LIN {X 0,Y 461.687,Z 311.629,A -85,B 0,C 180,E1 20728.292,E2 20728.292} C_VEL
LIN {X 0,Y 456.016,Z 403.282,A -85,B 0,C 180,E1 20726.276,E2 20726.276} C_VEL
LIN {X 0,Y 452.13,Z 492.328,A -85,B 0,C 180,E1 20724.472,E2 20724.472} C_VEL
LIN {X 0,Y 450.29,Z 542.964,A -85,B 0,C 180,E1 20723.46,E2 20723.46} C_VEL
LIN {X 0,Y 449.055,Z 565.43,A -85,B 0,C 180,E1 20722.774,E2 20722.774} C_VEL
LIN {X 0,Y 447.46,Z 585.999,A -85,B 0,C 180,E1 20721.912,E2 20721.912} C_VEL
LIN {X 0,Y 445.534,Z 606.342,A -85,B 0,C 180,E1 20720.838,E2 20720.838} C_VEL
LIN {X 0,Y 443.351,Z 625.885,A -85,B 0,C 180,E1 20719.568,E2 20719.568} C_VEL
LIN {X 0,Y 440.916,Z 645.179,A -85,B 0,C 180,E1 20718.033,E2 20718.033} C_VEL
LIN {X 0,Y 438.41,Z 662.746,A -85,B 0,C 180,E1 20716.361,E2 20716.361} C_VEL
LIN {X 0,Y 435.747,Z 680.551,A -85,B 0,C 180,E1 20714.35,E2 20714.35} C_VEL
LIN {X 0,Y 433.448,Z 695.322,A -85,B 0,C 180,E1 20712.389,E2 20712.389} C_VEL
LIN {X 0,Y 431.176,Z 709.526,A -85,B 0,C 180,E1 20710.152,E2 20710.152} C_VEL
LIN {X 0,Y 429.165,Z 722.41,A -85,B 0,C 180,E1 20707.768,E2 20707.768} C_VEL
LIN {X 0,Y 427.471,Z 733.989,A -85,B 0,C 180,E1 20705.236,E2 20705.236} C_VEL
LIN {X 0,Y 426.053,Z 744.612,A -85,B 0,C 180,E1 20702.423,E2 20702.423} C_VEL
LIN {X 0,Y 425.075,Z 753.264,A -85,B 0,C 180,E1 20699.598,E2 20699.598} C_VEL
LIN {X 0,Y 424.433,Z 760.513,A -85,B 0,C 180,E1 20696.626,E2 20696.626} C_VEL
LIN {X 0,Y 424.108,Z 766.032,A -85,B 0,C 180,E1 20693.64,E2 20693.64} C_VEL
LIN {X 0,Y 423.956,Z 769.849,A -85,B 0,C 180,E1 20690.637,E2 20690.637} C_VEL
LIN {X 0,Y 423.908,Z 772.115,A -85,B 0,C 180,E1 20687.554,E2 20687.554} C_VEL
LIN {X 0,Y 423.909,Z 772.685,A -85,B 0,C 180,E1 20684.685,E2 20684.685} C_VEL
LIN {X 0,Y 423.917,Z 771.748,A -85,B 0,C 180,E1 20681.72,E2 20681.72} C_VEL
LIN {X 0,Y 423.96,Z 769.376,A -85,B 0,C 180,E1 20678.851,E2 20678.851} C_VEL
LIN {X 0,Y 424.122,Z 765.205,A -85,B 0,C 180,E1 20675.833,E2 20675.833} C_VEL
LIN {X 0,Y 424.469,Z 759.552,A -85,B 0,C 180,E1 20672.925,E2 20672.925} C_VEL
LIN {X 0,Y 425.092,Z 752.337,A -85,B 0,C 180,E1 20670.092,E2 20670.092} C_VEL
LIN {X 0,Y 426.049,Z 743.659,A -85,B 0,C 180,E1 20667.335,E2 20667.335} C_VEL
LIN {X 0,Y 427.452,Z 732.887,A -85,B 0,C 180,E1 20664.546,E2 20664.546} C_VEL
LIN {X 0,Y 429.192,Z 720.789,A -85,B 0,C 180,E1 20661.946,E2 20661.946} C_VEL
LIN {X 0,Y 431.283,Z 707.328,A -85,B 0,C 180,E1 20659.502,E2 20659.502} C_VEL
LIN {X 0,Y 433.641,Z 692.685,A -85,B 0,C 180,E1 20657.235,E2 20657.235} C_VEL
LIN {X 0,Y 436.131,Z 676.972,A -85,B 0,C 180,E1 20655.177,E2 20655.177} C_VEL
LIN {X 0,Y 438.816,Z 659.657,A -85,B 0,C 180,E1 20653.251,E2 20653.251} C_VEL
LIN {X 0,Y 441.492,Z 641.523,A -85,B 0,C 180,E1 20651.54,E2 20651.54} C_VEL
LIN {X 0,Y 444.045,Z 622.624,A -85,B 0,C 180,E1 20650.046,E2 20650.046} C_VEL
LIN {X 0,Y 446.37,Z 603.344,A -85,B 0,C 180,E1 20648.789,E2 20648.789} C_VEL
LIN {X 0,Y 448.52,Z 582.74,A -85,B 0,C 180,E1 20647.69,E2 20647.69} C_VEL
LIN {X 0,Y 450.361,Z 560.984,A -85,B 0,C 180,E1 20646.784,E2 20646.784} C_VEL
LIN {X 0,Y 451.734,Z 539.486,A -85,B 0,C 180,E1 20646.135,E2 20646.135} C_VEL
LIN {X 0,Y 452.996,Z 507.273,A -85,B 0,C 180,E1 20645.485,E2 20645.485} C_VEL
LIN {X 0,Y 459.53,Z 311.984,A -85,B 0,C 180,E1 20641.902,E2 20641.902} C_VEL
LIN {X 0,Y 459.296,Z 310.719,A -85,B 0,C 180,E1 20641.847,E2 20641.847} C_VEL
LIN {X 0,Y 453.846,Z 302.158,A -85,B 0,C 180,E1 20641.015,E2 20641.015} C_VEL
LIN {X 0,Y 449.692,Z 297.638,A -85,B 0,C 180,E1 20640.411,E2 20640.411} C_VEL
LIN {X 0,Y 436.277,Z 287.787,A -85,B 0,C 180,E1 20638.475,E2 20638.475} C_VEL
LIN {X 0,Y 433.432,Z 284.546,A -85,B 0,C 180,E1 20638.01,E2 20638.01} C_VEL
LIN {X 0,Y 426.78,Z 275.226,A -85,B 0,C 180,E1 20636.846,E2 20636.846} C_VEL
LIN {X 0,Y 423.848,Z 271.045,A -85,B 0,C 180,E1 20636.316,E2 20636.316} C_VEL
LIN {X 0,Y 421.137,Z 267.04,A -85,B 0,C 180,E1 20635.81,E2 20635.81} C_VEL
LIN {X 0,Y 418.11,Z 263.221,A -85,B 0,C 180,E1 20635.251,E2 20635.251} C_VEL
LIN {X 0,Y 417.38,Z 260.741,A -85,B 0,C 180,E1 20635.046,E2 20635.046} C_VEL
LIN {X 0,Y 417.385,Z 260.741,A -85,B 0,C 180,E1 20631.207,E2 20631.207} C_VEL
LIN {X 0,Y 417.373,Z 260.747,A -85,B 0,C 180,E1 20627.282,E2 20627.282} C_VEL
LIN {X 0,Y 417.36,Z 260.74,A -85,B 0,C 180,E1 20623.438,E2 20623.438} C_VEL
LIN {X 0,Y 417.345,Z 260.748,A -85,B 0,C 180,E1 20619.656,E2 20619.656} C_VEL
LIN {X 0,Y 417.338,Z 260.742,A -85,B 0,C 180,E1 20615.914,E2 20615.914} C_VEL
LIN {X 0,Y 417.339,Z 260.741,A -85,B 0,C 180,E1 20612.061,E2 20612.061} C_VEL
LIN {X 0,Y 417.356,Z 260.741,A -85,B 0,C 180,E1 20608.354,E2 20608.354} C_VEL
LIN {X 0,Y 417.368,Z 260.74,A -85,B 0,C 180,E1 20604.503,E2 20604.503} C_VEL
LIN {X 0,Y 417.376,Z 260.74,A -85,B 0,C 180,E1 20600.724,E2 20600.724} C_VEL
LIN {X 0,Y 417.366,Z 260.742,A -85,B 0,C 180,E1 20596.847,E2 20596.847} C_VEL
LIN {X 0,Y 417.34,Z 260.744,A -85,B 0,C 180,E1 20593.15,E2 20593.15} C_VEL
LIN {X 0,Y 417.329,Z 260.745,A -85,B 0,C 180,E1 20589.38,E2 20589.38} C_VEL
LIN {X 0,Y 417.327,Z 260.745,A -85,B 0,C 180,E1 20585.515,E2 20585.515} C_VEL
LIN {X 0,Y 417.331,Z 260.743,A -85,B 0,C 180,E1 20581.683,E2 20581.683} C_VEL
LIN {X 0,Y 417.351,Z 260.742,A -85,B 0,C 180,E1 20577.998,E2 20577.998} C_VEL
LIN {X 0,Y 417.366,Z 260.747,A -85,B 0,C 180,E1 20574.232,E2 20574.232} C_VEL
LIN {X 0,Y 417.365,Z 260.751,A -85,B 0,C 180,E1 20570.416,E2 20570.416} C_VEL
LIN {X 0,Y 417.332,Z 260.751,A -85,B 0,C 180,E1 20566.743,E2 20566.743} C_VEL
LIN {X 0,Y 417.318,Z 260.749,A -85,B 0,C 180,E1 20563.053,E2 20563.053} C_VEL
LIN {X 0,Y 417.319,Z 260.744,A -85,B 0,C 180,E1 20559.233,E2 20559.233} C_VEL
LIN {X 0,Y 417.326,Z 260.743,A -85,B 0,C 180,E1 20555.433,E2 20555.433} C_VEL
LIN {X 0,Y 417.35,Z 260.747,A -85,B 0,C 180,E1 20551.74,E2 20551.74} C_VEL
LIN {X 0,Y 417.37,Z 260.749,A -85,B 0,C 180,E1 20547.878,E2 20547.878} C_VEL
LIN {X 0,Y 417.361,Z 260.747,A -85,B 0,C 180,E1 20543.88,E2 20543.88} C_VEL
LIN {X 0,Y 417.339,Z 260.747,A -85,B 0,C 180,E1 20540.097,E2 20540.097} C_VEL
LIN {X 0,Y 417.321,Z 260.75,A -85,B 0,C 180,E1 20536.277,E2 20536.277} C_VEL
LIN {X 0,Y 417.305,Z 260.752,A -85,B 0,C 180,E1 20532.591,E2 20532.591} C_VEL
LIN {X 0,Y 417.302,Z 260.753,A -85,B 0,C 180,E1 20528.68,E2 20528.68} C_VEL
LIN {X 0,Y 417.31,Z 260.751,A -85,B 0,C 180,E1 20524.946,E2 20524.946} C_VEL
LIN {X 0,Y 417.332,Z 260.746,A -85,B 0,C 180,E1 20521.234,E2 20521.234} C_VEL
LIN {X 0,Y 417.349,Z 260.745,A -85,B 0,C 180,E1 20517.527,E2 20517.527} C_VEL
LIN {X 0,Y 417.341,Z 260.746,A -85,B 0,C 180,E1 20513.671,E2 20513.671} C_VEL
LIN {X 0,Y 417.321,Z 260.752,A -85,B 0,C 180,E1 20509.926,E2 20509.926} C_VEL
LIN {X 0,Y 417.311,Z 260.747,A -85,B 0,C 180,E1 20506.136,E2 20506.136} C_VEL
LIN {X 0,Y 417.31,Z 260.751,A -85,B 0,C 180,E1 20502.283,E2 20502.283} C_VEL
LIN {X 0,Y 417.317,Z 260.747,A -85,B 0,C 180,E1 20498.494,E2 20498.494} C_VEL
LIN {X 0,Y 417.337,Z 260.745,A -85,B 0,C 180,E1 20494.756,E2 20494.756} C_VEL
LIN {X 0,Y 417.367,Z 260.744,A -85,B 0,C 180,E1 20490.971,E2 20490.971} C_VEL
LIN {X 0,Y 417.369,Z 260.745,A -85,B 0,C 180,E1 20487.056,E2 20487.056} C_VEL
LIN {X 0,Y 417.353,Z 260.9,A -85,B 0,C 180,E1 20484.489,E2 20484.489} C_VEL
LIN {X 0,Y 418.724,Z 264.377,A -85,B 0,C 180,E1 20483.856,E2 20483.856} C_VEL
LIN {X 0,Y 419.823,Z 266.306,A -85,B 0,C 180,E1 20483.457,E2 20483.457} C_VEL
LIN {X 0,Y 426.173,Z 279.213,A -85,B 0,C 180,E1 20481.04,E2 20481.04} C_VEL
LIN {X 0,Y 433.831,Z 295.144,A -85,B 0,C 180,E1 20478.323,E2 20478.323} C_VEL
LIN {X 0,Y 447.357,Z 317.125,A -85,B 0,C 180,E1 20475.986,E2 20475.986} C_VEL
LIN {X 0,Y 452.72,Z 326.557,A -85,B 0,C 180,E1 20475.107,E2 20475.107} C_VEL
LIN {X 0,Y 454.518,Z 340.457,A -85,B 0,C 180,E1 20474.557,E2 20474.557} C_VEL
LIN {X 0,Y 447.482,Z 532.078,A -85,B 0,C 180,E1 20470.954,E2 20470.954} C_VEL
LIN {X 0,Y 444.973,Z 604.939,A -85,B 0,C 180,E1 20469.579,E2 20469.579} C_VEL
LIN {X 0,Y 443.305,Z 627.558,A -85,B 0,C 180,E1 20468.939,E2 20468.939} C_VEL
LIN {X 0,Y 441.363,Z 648.539,A -85,B 0,C 180,E1 20468.118,E2 20468.118} C_VEL
LIN {X 0,Y 439.156,Z 668.895,A -85,B 0,C 180,E1 20467.108,E2 20467.108} C_VEL
LIN {X 0,Y 436.554,Z 689.548,A -85,B 0,C 180,E1 20465.827,E2 20465.827} C_VEL
LIN {X 0,Y 433.887,Z 708.868,A -85,B 0,C 180,E1 20464.371,E2 20464.371} C_VEL
LIN {X 0,Y 431.094,Z 728.01,A -85,B 0,C 180,E1 20462.655,E2 20462.655} C_VEL
LIN {X 0,Y 428.35,Z 746.056,A -85,B 0,C 180,E1 20460.741,E2 20460.741} C_VEL
LIN {X 0,Y 425.703,Z 762.95,A -85,B 0,C 180,E1 20458.627,E2 20458.627} C_VEL
LIN {X 0,Y 423.216,Z 779.4,A -85,B 0,C 180,E1 20456.216,E2 20456.216} C_VEL
LIN {X 0,Y 421.187,Z 793.532,A -85,B 0,C 180,E1 20453.799,E2 20453.799} C_VEL
LIN {X 0,Y 419.48,Z 806.214,A -85,B 0,C 180,E1 20451.24,E2 20451.24} C_VEL
LIN {X 0,Y 418.129,Z 817.539,A -85,B 0,C 180,E1 20448.543,E2 20448.543} C_VEL
LIN {X 0,Y 417.184,Z 827.072,A -85,B 0,C 180,E1 20445.854,E2 20445.854} C_VEL
LIN {X 0,Y 416.539,Z 835.158,A -85,B 0,C 180,E1 20443.039,E2 20443.039} C_VEL
LIN {X 0,Y 416.164,Z 841.833,A -85,B 0,C 180,E1 20440.1,E2 20440.1} C_VEL
LIN {X 0,Y 416.004,Z 846.599,A -85,B 0,C 180,E1 20437.317,E2 20437.317} C_VEL
LIN {X 0,Y 415.949,Z 849.714,A -85,B 0,C 180,E1 20434.548,E2 20434.548} C_VEL
LIN {X 0,Y 415.932,Z 851.456,A -85,B 0,C 180,E1 20431.789,E2 20431.789} C_VEL
LIN {X 0,Y 415.941,Z 851.599,A -85,B 0,C 180,E1 20429.034,E2 20429.034} C_VEL
LIN {X 0,Y 415.944,Z 850.257,A -85,B 0,C 180,E1 20426.139,E2 20426.139} C_VEL
LIN {X 0,Y 415.977,Z 847.555,A -85,B 0,C 180,E1 20423.512,E2 20423.512} C_VEL
LIN {X 0,Y 416.122,Z 842.982,A -85,B 0,C 180,E1 20420.595,E2 20420.595} C_VEL
LIN {X 0,Y 416.422,Z 836.946,A -85,B 0,C 180,E1 20417.801,E2 20417.801} C_VEL
LIN {X 0,Y 416.999,Z 828.674,A -85,B 0,C 180,E1 20414.848,E2 20414.848} C_VEL
LIN {X 0,Y 417.889,Z 818.824,A -85,B 0,C 180,E1 20412.021,E2 20412.021} C_VEL
LIN {X 0,Y 419.112,Z 807.467,A -85,B 0,C 180,E1 20409.323,E2 20409.323} C_VEL
LIN {X 0,Y 420.647,Z 794.563,A -85,B 0,C 180,E1 20406.759,E2 20406.759} C_VEL
LIN {X 0,Y 422.49,Z 780.254,A -85,B 0,C 180,E1 20404.335,E2 20404.335} C_VEL
LIN {X 0,Y 424.623,Z 764.525,A -85,B 0,C 180,E1 20402.056,E2 20402.056} C_VEL
LIN {X 0,Y 426.972,Z 747.129,A -85,B 0,C 180,E1 20399.924,E2 20399.924} C_VEL
LIN {X 0,Y 429.494,Z 728.046,A -85,B 0,C 180,E1 20397.93,E2 20397.93} C_VEL
LIN {X 0,Y 432.046,Z 708.264,A -85,B 0,C 180,E1 20396.183,E2 20396.183} C_VEL
LIN {X 0,Y 434.455,Z 688.453,A -85,B 0,C 180,E1 20394.713,E2 20394.713} C_VEL
LIN {X 0,Y 436.862,Z 666.955,A -85,B 0,C 180,E1 20393.4,E2 20393.4} C_VEL
LIN {X 0,Y 439.103,Z 644.338,A -85,B 0,C 180,E1 20392.284,E2 20392.284} C_VEL
LIN {X 0,Y 441.135,Z 621.158,A -85,B 0,C 180,E1 20391.4,E2 20391.4} C_VEL
LIN {X 0,Y 442.81,Z 597.262,A -85,B 0,C 180,E1 20390.738,E2 20390.738} C_VEL
LIN {X 0,Y 447.425,Z 477.005,A -85,B 0,C 180,E1 20388.341,E2 20388.341} C_VEL
LIN {X 0,Y 452.446,Z 386.097,A -85,B 0,C 180,E1 20386.36,E2 20386.36} C_VEL
LIN {X 0,Y 455.647,Z 338.78,A -85,B 0,C 180,E1 20385.25,E2 20385.25} C_VEL
LIN {X 0,Y 454.596,Z 324.963,A -85,B 0,C 180,E1 20384.558,E2 20384.558} C_VEL
LIN {X 0,Y 449.935,Z 312.613,A -85,B 0,C 180,E1 20383.128,E2 20383.128} C_VEL
LIN {X 0,Y 446.26,Z 303.945,A -85,B 0,C 180,E1 20381.756,E2 20381.756} C_VEL
LIN {X 0,Y 443.328,Z 297.389,A -85,B 0,C 180,E1 20380.338,E2 20380.338} C_VEL
LIN {X 0,Y 441.972,Z 294.021,A -85,B 0,C 180,E1 20379.389,E2 20379.389} C_VEL
LIN {X 0,Y 440.851,Z 290.72,A -85,B 0,C 180,E1 20378.091,E2 20378.091} C_VEL
LIN {X 0,Y 440.662,Z 288.86,A -85,B 0,C 180,E1 20376.315,E2 20376.315} C_VEL
LIN {X 0,Y 441.578,Z 288.676,A -85,B 0,C 180,E1 20375.11,E2 20375.11} C_VEL
LIN {X 0,Y 443.459,Z 292.182,A -85,B 0,C 180,E1 20373.568,E2 20373.568} C_VEL
LIN {X 0,Y 444.508,Z 293.515,A -85,B 0,C 180,E1 20373.028,E2 20373.028} C_VEL
LIN {X 0,Y 447.412,Z 298.49,A -85,B 0,C 180,E1 20371.752,E2 20371.752} C_VEL
LIN {X 0,Y 450.394,Z 303.654,A -85,B 0,C 180,E1 20370.724,E2 20370.724} C_VEL
LIN {X 0,Y 454.787,Z 311.649,A -85,B 0,C 180,E1 20369.469,E2 20369.469} C_VEL
LIN {X 0,Y 456.507,Z 315.582,A -85,B 0,C 180,E1 20368.999,E2 20368.999} C_VEL
LIN {X 0,Y 450.521,Z 400.716,A -85,B 0,C 180,E1 20367.055,E2 20367.055} C_VEL
LIN {X 0,Y 446.275,Z 483.639,A -85,B 0,C 180,E1 20365.293,E2 20365.293} C_VEL
LIN {X 0,Y 443.839,Z 544.168,A -85,B 0,C 180,E1 20364.051,E2 20364.051} C_VEL
LIN {X 0,Y 442.514,Z 566.682,A -85,B 0,C 180,E1 20363.346,E2 20363.346} C_VEL
LIN {X 0,Y 440.774,Z 587.885,A -85,B 0,C 180,E1 20362.438,E2 20362.438} C_VEL
LIN {X 0,Y 438.676,Z 608.667,A -85,B 0,C 180,E1 20361.308,E2 20361.308} C_VEL
LIN {X 0,Y 436.301,Z 628.61,A -85,B 0,C 180,E1 20359.967,E2 20359.967} C_VEL
LIN {X 0,Y 433.87,Z 646.94,A -85,B 0,C 180,E1 20358.475,E2 20358.475} C_VEL
LIN {X 0,Y 431.127,Z 665.128,A -85,B 0,C 180,E1 20356.699,E2 20356.699} C_VEL
LIN {X 0,Y 428.451,Z 682.036,A -85,B 0,C 180,E1 20354.738,E2 20354.738} C_VEL
LIN {X 0,Y 425.88,Z 697.593,A -85,B 0,C 180,E1 20352.613,E2 20352.613} C_VEL
LIN {X 0,Y 423.532,Z 711.677,A -85,B 0,C 180,E1 20350.337,E2 20350.337} C_VEL
LIN {X 0,Y 421.432,Z 724.354,A -85,B 0,C 180,E1 20347.911,E2 20347.911} C_VEL
LIN {X 0,Y 419.664,Z 735.756,A -85,B 0,C 180,E1 20345.333,E2 20345.333} C_VEL
LIN {X 0,Y 418.253,Z 745.811,A -85,B 0,C 180,E1 20342.605,E2 20342.605} C_VEL
LIN {X 0,Y 417.21,Z 754.395,A -85,B 0,C 180,E1 20339.727,E2 20339.727} C_VEL
LIN {X 0,Y 416.522,Z 761.571,A -85,B 0,C 180,E1 20336.699,E2 20336.699} C_VEL
LIN {X 0,Y 416.183,Z 766.824,A -85,B 0,C 180,E1 20333.796,E2 20333.796} C_VEL
LIN {X 0,Y 416.005,Z 770.638,A -85,B 0,C 180,E1 20330.735,E2 20330.735} C_VEL
LIN {X 0,Y 415.944,Z 772.843,A -85,B 0,C 180,E1 20327.649,E2 20327.649} C_VEL
LIN {X 0,Y 415.944,Z 773.434,A -85,B 0,C 180,E1 20324.67,E2 20324.67} C_VEL
LIN {X 0,Y 415.954,Z 772.467,A -85,B 0,C 180,E1 20321.648,E2 20321.648} C_VEL
LIN {X 0,Y 416.001,Z 770.04,A -85,B 0,C 180,E1 20318.722,E2 20318.722} C_VEL
LIN {X 0,Y 416.182,Z 766.014,A -85,B 0,C 180,E1 20315.746,E2 20315.746} C_VEL
LIN {X 0,Y 416.569,Z 760.212,A -85,B 0,C 180,E1 20312.716,E2 20312.716} C_VEL
LIN {X 0,Y 417.261,Z 752.848,A -85,B 0,C 180,E1 20309.79,E2 20309.79} C_VEL
LIN {X 0,Y 418.301,Z 744.086,A -85,B 0,C 180,E1 20306.98,E2 20306.98} C_VEL
LIN {X 0,Y 419.821,Z 733.267,A -85,B 0,C 180,E1 20304.138,E2 20304.138} C_VEL
LIN {X 0,Y 421.6,Z 721.552,A -85,B 0,C 180,E1 20301.588,E2 20301.588} C_VEL
LIN {X 0,Y 423.907,Z 707.522,A -85,B 0,C 180,E1 20299.007,E2 20299.007} C_VEL
LIN {X 0,Y 426.419,Z 692.741,A -85,B 0,C 180,E1 20296.701,E2 20296.701} C_VEL
LIN {X 0,Y 429.059,Z 676.948,A -85,B 0,C 180,E1 20294.612,E2 20294.612} C_VEL
LIN {X 0,Y 431.797,Z 660.122,A -85,B 0,C 180,E1 20292.725,E2 20292.725} C_VEL
LIN {X 0,Y 434.638,Z 641.692,A -85,B 0,C 180,E1 20290.968,E2 20290.968} C_VEL
LIN {X 0,Y 437.408,Z 622.143,A -85,B 0,C 180,E1 20289.414,E2 20289.414} C_VEL
LIN {X 0,Y 439.835,Z 602.544,A -85,B 0,C 180,E1 20288.141,E2 20288.141} C_VEL
LIN {X 0,Y 442.167,Z 580.437,A -85,B 0,C 180,E1 20286.978,E2 20286.978} C_VEL
LIN {X 0,Y 444.072,Z 558.464,A -85,B 0,C 180,E1 20286.089,E2 20286.089} C_VEL
LIN {X 0,Y 445.45,Z 537.35,A -85,B 0,C 180,E1 20285.466,E2 20285.466} C_VEL
LIN {X 0,Y 447.035,Z 494.669,A -85,B 0,C 180,E1 20284.632,E2 20284.632} C_VEL
LIN {X 0,Y 453.499,Z 314.519,A -85,B 0,C 180,E1 20281.263,E2 20281.263} C_VEL
LIN {X 0,Y 440.373,Z 294.525,A -85,B 0,C 180,E1 20279.183,E2 20279.183} C_VEL
LIN {X 0,Y 433.432,Z 284.546,A -85,B 0,C 180,E1 20278.01,E2 20278.01} C_VEL
LIN {X 0,Y 430.533,Z 281.967,A -85,B 0,C 180,E1 20277.547,E2 20277.547} C_VEL
LIN {X 0,Y 420.772,Z 277.941,A -85,B 0,C 180,E1 20276.074,E2 20276.074} C_VEL
LIN {X 0,Y 418.753,Z 276.061,A -85,B 0,C 180,E1 20275.725,E2 20275.725} C_VEL
LIN {X 0,Y 416.079,Z 272.148,A -85,B 0,C 180,E1 20275.211,E2 20275.211} C_VEL
LIN {X 0,Y 413.38,Z 268.174,A -85,B 0,C 180,E1 20274.68,E2 20274.68} C_VEL
LIN {X 0,Y 412.234,Z 266.897,A -85,B 0,C 180,E1 20274.467,E2 20274.467} C_VEL
LIN {X 0,Y 410.068,Z 264.072,A -85,B 0,C 180,E1 20274.049,E2 20274.049} C_VEL
LIN {X 0,Y 409.413,Z 261.738,A -85,B 0,C 180,E1 20273.841,E2 20273.841} C_VEL
LIN {X 0,Y 409.406,Z 261.738,A -85,B 0,C 180,E1 20269.994,E2 20269.994} C_VEL
LIN {X 0,Y 409.403,Z 261.734,A -85,B 0,C 180,E1 20266.021,E2 20266.021} C_VEL
LIN {X 0,Y 409.403,Z 261.737,A -85,B 0,C 180,E1 20262.125,E2 20262.125} C_VEL
LIN {X 0,Y 409.409,Z 261.731,A -85,B 0,C 180,E1 20258.286,E2 20258.286} C_VEL
LIN {X 0,Y 409.422,Z 261.732,A -85,B 0,C 180,E1 20254.483,E2 20254.483} C_VEL
LIN {X 0,Y 409.433,Z 261.733,A -85,B 0,C 180,E1 20250.561,E2 20250.561} C_VEL
LIN {X 0,Y 409.433,Z 261.728,A -85,B 0,C 180,E1 20246.641,E2 20246.641} C_VEL
LIN {X 0,Y 409.449,Z 261.725,A -85,B 0,C 180,E1 20242.706,E2 20242.706} C_VEL
LIN {X 0,Y 409.432,Z 261.727,A -85,B 0,C 180,E1 20238.736,E2 20238.736} C_VEL
LIN {X 0,Y 409.423,Z 261.729,A -85,B 0,C 180,E1 20234.854,E2 20234.854} C_VEL
LIN {X 0,Y 409.405,Z 261.734,A -85,B 0,C 180,E1 20231.047,E2 20231.047} C_VEL
LIN {X 0,Y 409.391,Z 261.736,A -85,B 0,C 180,E1 20227.303,E2 20227.303} C_VEL
LIN {X 0,Y 409.39,Z 261.737,A -85,B 0,C 180,E1 20223.359,E2 20223.359} C_VEL
LIN {X 0,Y 409.388,Z 261.74,A -85,B 0,C 180,E1 20219.471,E2 20219.471} C_VEL
LIN {X 0,Y 409.392,Z 261.742,A -85,B 0,C 180,E1 20215.634,E2 20215.634} C_VEL
LIN {X 0,Y 409.407,Z 261.738,A -85,B 0,C 180,E1 20211.841,E2 20211.841} C_VEL
LIN {X 0,Y 409.432,Z 261.73,A -85,B 0,C 180,E1 20208.14,E2 20208.14} C_VEL
LIN {X 0,Y 409.42,Z 261.732,A -85,B 0,C 180,E1 20204.299,E2 20204.299} C_VEL
LIN {X 0,Y 409.414,Z 261.737,A -85,B 0,C 180,E1 20200.366,E2 20200.366} C_VEL
LIN {X 0,Y 409.393,Z 261.741,A -85,B 0,C 180,E1 20196.536,E2 20196.536} C_VEL
LIN {X 0,Y 409.378,Z 261.74,A -85,B 0,C 180,E1 20192.831,E2 20192.831} C_VEL
LIN {X 0,Y 409.374,Z 261.738,A -85,B 0,C 180,E1 20188.918,E2 20188.918} C_VEL
LIN {X 0,Y 409.373,Z 261.735,A -85,B 0,C 180,E1 20184.992,E2 20184.992} C_VEL
LIN {X 0,Y 409.38,Z 261.736,A -85,B 0,C 180,E1 20181.188,E2 20181.188} C_VEL
LIN {X 0,Y 409.4,Z 261.734,A -85,B 0,C 180,E1 20177.479,E2 20177.479} C_VEL
LIN {X 0,Y 409.416,Z 261.733,A -85,B 0,C 180,E1 20173.605,E2 20173.605} C_VEL
LIN {X 0,Y 409.41,Z 261.735,A -85,B 0,C 180,E1 20169.699,E2 20169.699} C_VEL
LIN {X 0,Y 409.395,Z 261.738,A -85,B 0,C 180,E1 20165.885,E2 20165.885} C_VEL
LIN {X 0,Y 409.376,Z 261.742,A -85,B 0,C 180,E1 20162.098,E2 20162.098} C_VEL
LIN {X 0,Y 409.366,Z 261.741,A -85,B 0,C 180,E1 20158.319,E2 20158.319} C_VEL
LIN {X 0,Y 409.366,Z 261.735,A -85,B 0,C 180,E1 20154.392,E2 20154.392} C_VEL
LIN {X 0,Y 409.369,Z 261.741,A -85,B 0,C 180,E1 20150.438,E2 20150.438} C_VEL
LIN {X 0,Y 409.374,Z 261.736,A -85,B 0,C 180,E1 20146.582,E2 20146.582} C_VEL
LIN {X 0,Y 409.402,Z 261.737,A -85,B 0,C 180,E1 20142.957,E2 20142.957} C_VEL
LIN {X 0,Y 409.422,Z 261.731,A -85,B 0,C 180,E1 20139.11,E2 20139.11} C_VEL
LIN {X 0,Y 409.418,Z 261.736,A -85,B 0,C 180,E1 20135.291,E2 20135.291} C_VEL
LIN {X 0,Y 409.409,Z 261.738,A -85,B 0,C 180,E1 20131.4,E2 20131.4} C_VEL
LIN {X 0,Y 409.389,Z 261.742,A -85,B 0,C 180,E1 20127.664,E2 20127.664} C_VEL
LIN {X 0,Y 409.404,Z 261.861,A -85,B 0,C 180,E1 20125.655,E2 20125.655} C_VEL
LIN {X 0,Y 410.549,Z 264.935,A -85,B 0,C 180,E1 20125.086,E2 20125.086} C_VEL
LIN {X 0,Y 411.698,Z 266.708,A -85,B 0,C 180,E1 20124.685,E2 20124.685} C_VEL
LIN {X 0,Y 413.768,Z 270.754,A -85,B 0,C 180,E1 20123.869,E2 20123.869} C_VEL
LIN {X 0,Y 422.506,Z 288.809,A -85,B 0,C 180,E1 20120.484,E2 20120.484} C_VEL
LIN {X 0,Y 425.258,Z 294.502,A -85,B 0,C 180,E1 20119.538,E2 20119.538} C_VEL
LIN {X 0,Y 438.285,Z 315.212,A -85,B 0,C 180,E1 20117.191,E2 20117.191} C_VEL
LIN {X 0,Y 447.194,Z 330.714,A -85,B 0,C 180,E1 20115.669,E2 20115.669} C_VEL
LIN {X 0,Y 448.597,Z 341.984,A -85,B 0,C 180,E1 20115.223,E2 20115.223} C_VEL
LIN {X 0,Y 441.022,Z 536.438,A -85,B 0,C 180,E1 20111.51,E2 20111.51} C_VEL
LIN {X 0,Y 438.534,Z 604.38,A -85,B 0,C 180,E1 20110.204,E2 20110.204} C_VEL
LIN {X 0,Y 436.767,Z 627.096,A -85,B 0,C 180,E1 20109.554,E2 20109.554} C_VEL
LIN {X 0,Y 434.724,Z 648.068,A -85,B 0,C 180,E1 20108.724,E2 20108.724} C_VEL
LIN {X 0,Y 432.26,Z 669.526,A -85,B 0,C 180,E1 20107.635,E2 20107.635} C_VEL
LIN {X 0,Y 429.583,Z 689.731,A -85,B 0,C 180,E1 20106.358,E2 20106.358} C_VEL
LIN {X 0,Y 426.752,Z 709.126,A -85,B 0,C 180,E1 20104.865,E2 20104.865} C_VEL
LIN {X 0,Y 423.68,Z 729.071,A -85,B 0,C 180,E1 20103.032,E2 20103.032} C_VEL
LIN {X 0,Y 420.829,Z 746.97,A -85,B 0,C 180,E1 20101.088,E2 20101.088} C_VEL
LIN {X 0,Y 418.013,Z 764.019,A -85,B 0,C 180,E1 20098.891,E2 20098.891} C_VEL
LIN {X 0,Y 415.562,Z 779.308,A -85,B 0,C 180,E1 20096.583,E2 20096.583} C_VEL
LIN {X 0,Y 413.428,Z 793.348,A -85,B 0,C 180,E1 20094.123,E2 20094.123} C_VEL
LIN {X 0,Y 411.634,Z 805.994,A -85,B 0,C 180,E1 20091.515,E2 20091.515} C_VEL
LIN {X 0,Y 410.214,Z 817.242,A -85,B 0,C 180,E1 20088.766,E2 20088.766} C_VEL
LIN {X 0,Y 409.187,Z 827.129,A -85,B 0,C 180,E1 20085.881,E2 20085.881} C_VEL
LIN {X 0,Y 408.545,Z 834.946,A -85,B 0,C 180,E1 20083.079,E2 20083.079} C_VEL
LIN {X 0,Y 408.179,Z 841.351,A -85,B 0,C 180,E1 20080.157,E2 20080.157} C_VEL
LIN {X 0,Y 408.021,Z 846.062,A -85,B 0,C 180,E1 20077.319,E2 20077.319} C_VEL
LIN {X 0,Y 407.974,Z 849.102,A -85,B 0,C 180,E1 20074.497,E2 20074.497} C_VEL
LIN {X 0,Y 407.966,Z 850.771,A -85,B 0,C 180,E1 20071.543,E2 20071.543} C_VEL
LIN {X 0,Y 407.976,Z 850.825,A -85,B 0,C 180,E1 20068.875,E2 20068.875} C_VEL
LIN {X 0,Y 407.977,Z 849.35,A -85,B 0,C 180,E1 20065.923,E2 20065.923} C_VEL
LIN {X 0,Y 408.017,Z 846.566,A -85,B 0,C 180,E1 20063.244,E2 20063.244} C_VEL
LIN {X 0,Y 408.161,Z 841.832,A -85,B 0,C 180,E1 20060.267,E2 20060.267} C_VEL
LIN {X 0,Y 408.48,Z 835.655,A -85,B 0,C 180,E1 20057.416,E2 20057.416} C_VEL
LIN {X 0,Y 409.079,Z 827.627,A -85,B 0,C 180,E1 20054.548,E2 20054.548} C_VEL
LIN {X 0,Y 410.017,Z 817.692,A -85,B 0,C 180,E1 20051.664,E2 20051.664} C_VEL
LIN {X 0,Y 411.316,Z 806.225,A -85,B 0,C 180,E1 20048.913,E2 20048.913} C_VEL
LIN {X 0,Y 412.95,Z 793.188,A -85,B 0,C 180,E1 20046.3,E2 20046.3} C_VEL
LIN {X 0,Y 414.948,Z 778.379,A -85,B 0,C 180,E1 20043.778,E2 20043.778} C_VEL
LIN {X 0,Y 417.216,Z 762.272,A -85,B 0,C 180,E1 20041.437,E2 20041.437} C_VEL
LIN {X 0,Y 419.669,Z 745.147,A -85,B 0,C 180,E1 20039.327,E2 20039.327} C_VEL
LIN {X 0,Y 422.324,Z 726.13,A -85,B 0,C 180,E1 20037.329,E2 20037.329} C_VEL
LIN {X 0,Y 425.063,Z 705.689,A -85,B 0,C 180,E1 20035.522,E2 20035.522} C_VEL
LIN {X 0,Y 427.593,Z 686.093,A -85,B 0,C 180,E1 20034.06,E2 20034.06} C_VEL
LIN {X 0,Y 430.146,Z 664.332,A -85,B 0,C 180,E1 20032.732,E2 20032.732} C_VEL
LIN {X 0,Y 432.493,Z 641.784,A -85,B 0,C 180,E1 20031.621,E2 20031.621} C_VEL
LIN {X 0,Y 434.738,Z 617.66,A -85,B 0,C 180,E1 20030.713,E2 20030.713} C_VEL
LIN {X 0,Y 436.411,Z 594.283,A -85,B 0,C 180,E1 20030.068,E2 20030.068} C_VEL
LIN {X 0,Y 441.188,Z 482.742,A -85,B 0,C 180,E1 20027.77,E2 20027.77} C_VEL
LIN {X 0,Y 446.563,Z 394.596,A -85,B 0,C 180,E1 20025.787,E2 20025.787} C_VEL
LIN {X 0,Y 450.676,Z 340.484,A -85,B 0,C 180,E1 20024.477,E2 20024.477} C_VEL
LIN {X 0,Y 450.019,Z 329.12,A -85,B 0,C 180,E1 20023.885,E2 20023.885} C_VEL
LIN {X 0,Y 446.098,Z 317.872,A -85,B 0,C 180,E1 20022.506,E2 20022.506} C_VEL
LIN {X 0,Y 443.193,Z 310.242,A -85,B 0,C 180,E1 20021.25,E2 20021.25} C_VEL
LIN {X 0,Y 440.819,Z 304.2,A -85,B 0,C 180,E1 20019.892,E2 20019.892} C_VEL
LIN {X 0,Y 439.722,Z 301.042,A -85,B 0,C 180,E1 20018.953,E2 20018.953} C_VEL
LIN {X 0,Y 438.979,Z 298.236,A -85,B 0,C 180,E1 20017.786,E2 20017.786} C_VEL
LIN {X 0,Y 439.118,Z 296.576,A -85,B 0,C 180,E1 20016.066,E2 20016.066} C_VEL
LIN {X 0,Y 439.791,Z 296.658,A -85,B 0,C 180,E1 20015.194,E2 20015.194} C_VEL
LIN {X 0,Y 441.533,Z 299.894,A -85,B 0,C 180,E1 20013.699,E2 20013.699} C_VEL
LIN {X 0,Y 442.386,Z 301.375,A -85,B 0,C 180,E1 20013.195,E2 20013.195} C_VEL
LIN {X 0,Y 444.782,Z 305.722,A -85,B 0,C 180,E1 20012.06,E2 20012.06} C_VEL
LIN {X 0,Y 448.074,Z 311.755,A -85,B 0,C 180,E1 20010.85,E2 20010.85} C_VEL
LIN {X 0,Y 451.646,Z 319.134,A -85,B 0,C 180,E1 20009.751,E2 20009.751} C_VEL
LIN {X 0,Y 445.305,Z 397.926,A -85,B 0,C 180,E1 20007.879,E2 20007.879} C_VEL
LIN {X 0,Y 440.565,Z 477.774,A -85,B 0,C 180,E1 20006.105,E2 20006.105} C_VEL
LIN {X 0,Y 437.479,Z 545.67,A -85,B 0,C 180,E1 20004.662,E2 20004.662} C_VEL
LIN {X 0,Y 436.053,Z 568.238,A -85,B 0,C 180,E1 20003.933,E2 20003.933} C_VEL
LIN {X 0,Y 434.215,Z 589.312,A -85,B 0,C 180,E1 20003.011,E2 20003.011} C_VEL
LIN {X 0,Y 431.975,Z 610.202,A -85,B 0,C 180,E1 20001.848,E2 20001.848} C_VEL
LIN {X 0,Y 429.409,Z 630.62,A -85,B 0,C 180,E1 20000.444,E2 20000.444} C_VEL
LIN {X 0,Y 426.864,Z 648.771,A -85,B 0,C 180,E1 19998.931,E2 19998.931} C_VEL
LIN {X 0,Y 424.118,Z 666.053,A -85,B 0,C 180,E1 19997.211,E2 19997.211} C_VEL
LIN {X 0,Y 421.267,Z 683.105,A -85,B 0,C 180,E1 19995.2,E2 19995.2} C_VEL
LIN {X 0,Y 418.653,Z 698.174,A -85,B 0,C 180,E1 19993.115,E2 19993.115} C_VEL
LIN {X 0,Y 416.152,Z 712.264,A -85,B 0,C 180,E1 19990.803,E2 19990.803} C_VEL
LIN {X 0,Y 413.925,Z 725.017,A -85,B 0,C 180,E1 19988.335,E2 19988.335} C_VEL
LIN {X 0,Y 412.034,Z 736.456,A -85,B 0,C 180,E1 19985.712,E2 19985.712} C_VEL
LIN {X 0,Y 410.52,Z 746.539,A -85,B 0,C 180,E1 19982.934,E2 19982.934} C_VEL
LIN {X 0,Y 409.434,Z 754.775,A -85,B 0,C 180,E1 19980.142,E2 19980.142} C_VEL
LIN {X 0,Y 408.66,Z 762.064,A -85,B 0,C 180,E1 19977.057,E2 19977.057} C_VEL
LIN {X 0,Y 408.268,Z 767.396,A -85,B 0,C 180,E1 19974.098,E2 19974.098} C_VEL
LIN {X 0,Y 408.06,Z 771.116,A -85,B 0,C 180,E1 19971.122,E2 19971.122} C_VEL
LIN {X 0,Y 407.984,Z 773.497,A -85,B 0,C 180,E1 19967.919,E2 19967.919} C_VEL
LIN {X 0,Y 407.987,Z 774.211,A -85,B 0,C 180,E1 19964.926,E2 19964.926} C_VEL
LIN {X 0,Y 407.985,Z 773.385,A -85,B 0,C 180,E1 19961.969,E2 19961.969} C_VEL
LIN {X 0,Y 408.04,Z 771.038,A -85,B 0,C 180,E1 19958.89,E2 19958.89} C_VEL
LIN {X 0,Y 408.219,Z 767.147,A -85,B 0,C 180,E1 19955.858,E2 19955.858} C_VEL
LIN {X 0,Y 408.59,Z 761.758,A -85,B 0,C 180,E1 19952.928,E2 19952.928} C_VEL
LIN {X 0,Y 409.32,Z 754.4,A -85,B 0,C 180,E1 19949.853,E2 19949.853} C_VEL
LIN {X 0,Y 410.421,Z 745.639,A -85,B 0,C 180,E1 19946.93,E2 19946.93} C_VEL
LIN {X 0,Y 411.9,Z 735.454,A -85,B 0,C 180,E1 19944.172,E2 19944.172} C_VEL
LIN {X 0,Y 413.844,Z 723.407,A -85,B 0,C 180,E1 19941.443,E2 19941.443} C_VEL
LIN {X 0,Y 416.078,Z 710.6,A -85,B 0,C 180,E1 19938.988,E2 19938.988} C_VEL
LIN {X 0,Y 418.639,Z 696.126,A -85,B 0,C 180,E1 19936.638,E2 19936.638} C_VEL
LIN {X 0,Y 421.346,Z 680.756,A -85,B 0,C 180,E1 19934.517,E2 19934.517} C_VEL
LIN {X 0,Y 424.195,Z 664.26,A -85,B 0,C 180,E1 19932.57,E2 19932.57} C_VEL
LIN {X 0,Y 427.141,Z 646.239,A -85,B 0,C 180,E1 19930.776,E2 19930.776} C_VEL
LIN {X 0,Y 429.945,Z 627.336,A -85,B 0,C 180,E1 19929.199,E2 19929.199} C_VEL
LIN {X 0,Y 432.782,Z 606.315,A -85,B 0,C 180,E1 19927.752,E2 19927.752} C_VEL
LIN {X 0,Y 435.125,Z 586.329,A -85,B 0,C 180,E1 19926.633,E2 19926.633} C_VEL
LIN {X 0,Y 437.159,Z 564.343,A -85,B 0,C 180,E1 19925.673,E2 19925.673} C_VEL
LIN {X 0,Y 438.753,Z 542.399,A -85,B 0,C 180,E1 19924.967,E2 19924.967} C_VEL
LIN {X 0,Y 439.965,Z 516.998,A -85,B 0,C 180,E1 19924.411,E2 19924.411} C_VEL
LIN {X 0,Y 447.478,Z 317.982,A -85,B 0,C 180,E1 19920.645,E2 19920.645} C_VEL
LIN {X 0,Y 433.443,Z 296.639,A -85,B 0,C 180,E1 19918.336,E2 19918.336} C_VEL
LIN {X 0,Y 419.654,Z 277.152,A -85,B 0,C 180,E1 19915.889,E2 19915.889} C_VEL
LIN {X 0,Y 418.753,Z 276.061,A -85,B 0,C 180,E1 19915.725,E2 19915.725} C_VEL
LIN {X 0,Y 415.529,Z 273.23,A -85,B 0,C 180,E1 19915.161,E2 19915.161} C_VEL
LIN {X 0,Y 405.3,Z 268.606,A -85,B 0,C 180,E1 19913.443,E2 19913.443} C_VEL
LIN {X 0,Y 404.457,Z 267.986,A -85,B 0,C 180,E1 19913.288,E2 19913.288} C_VEL
LIN {X 0,Y 402.18,Z 265.102,A -85,B 0,C 180,E1 19912.821,E2 19912.821} C_VEL
LIN {X 0,Y 401.48,Z 262.723,A -85,B 0,C 180,E1 19912.592,E2 19912.592} C_VEL
LIN {X 0,Y 401.491,Z 262.719,A -85,B 0,C 180,E1 19908.74,E2 19908.74} C_VEL
LIN {X 0,Y 401.506,Z 262.723,A -85,B 0,C 180,E1 19904.864,E2 19904.864} C_VEL
LIN {X 0,Y 401.498,Z 262.718,A -85,B 0,C 180,E1 19900.911,E2 19900.911} C_VEL
LIN {X 0,Y 401.51,Z 262.722,A -85,B 0,C 180,E1 19896.866,E2 19896.866} C_VEL
LIN {X 0,Y 401.497,Z 262.716,A -85,B 0,C 180,E1 19892.856,E2 19892.856} C_VEL
LIN {X 0,Y 401.502,Z 262.711,A -85,B 0,C 180,E1 19888.86,E2 19888.86} C_VEL
LIN {X 0,Y 401.494,Z 262.712,A -85,B 0,C 180,E1 19884.858,E2 19884.858} C_VEL
LIN {X 0,Y 401.483,Z 262.716,A -85,B 0,C 180,E1 19880.975,E2 19880.975} C_VEL
LIN {X 0,Y 401.474,Z 262.72,A -85,B 0,C 180,E1 19877.049,E2 19877.049} C_VEL
LIN {X 0,Y 401.461,Z 262.722,A -85,B 0,C 180,E1 19873.209,E2 19873.209} C_VEL
LIN {X 0,Y 401.455,Z 262.722,A -85,B 0,C 180,E1 19869.29,E2 19869.29} C_VEL
LIN {X 0,Y 401.451,Z 262.722,A -85,B 0,C 180,E1 19865.37,E2 19865.37} C_VEL
LIN {X 0,Y 401.448,Z 262.721,A -85,B 0,C 180,E1 19861.434,E2 19861.434} C_VEL
LIN {X 0,Y 401.45,Z 262.719,A -85,B 0,C 180,E1 19857.593,E2 19857.593} C_VEL
LIN {X 0,Y 401.462,Z 262.721,A -85,B 0,C 180,E1 19853.793,E2 19853.793} C_VEL
LIN {X 0,Y 401.484,Z 262.726,A -85,B 0,C 180,E1 19850.022,E2 19850.022} C_VEL
LIN {X 0,Y 401.487,Z 262.73,A -85,B 0,C 180,E1 19846.188,E2 19846.188} C_VEL
LIN {X 0,Y 401.484,Z 262.726,A -85,B 0,C 180,E1 19842.249,E2 19842.249} C_VEL
LIN {X 0,Y 401.474,Z 262.721,A -85,B 0,C 180,E1 19838.322,E2 19838.322} C_VEL
LIN {X 0,Y 401.457,Z 262.718,A -85,B 0,C 180,E1 19834.424,E2 19834.424} C_VEL
LIN {X 0,Y 401.44,Z 262.724,A -85,B 0,C 180,E1 19830.7,E2 19830.7} C_VEL
LIN {X 0,Y 401.437,Z 262.726,A -85,B 0,C 180,E1 19826.793,E2 19826.793} C_VEL
LIN {X 0,Y 401.434,Z 262.728,A -85,B 0,C 180,E1 19822.849,E2 19822.849} C_VEL
LIN {X 0,Y 401.432,Z 262.728,A -85,B 0,C 180,E1 19818.837,E2 19818.837} C_VEL
LIN {X 0,Y 401.428,Z 262.727,A -85,B 0,C 180,E1 19814.863,E2 19814.863} C_VEL
LIN {X 0,Y 401.436,Z 262.724,A -85,B 0,C 180,E1 19811.055,E2 19811.055} C_VEL
LIN {X 0,Y 401.453,Z 262.724,A -85,B 0,C 180,E1 19807.295,E2 19807.295} C_VEL
LIN {X 0,Y 401.464,Z 262.724,A -85,B 0,C 180,E1 19803.425,E2 19803.425} C_VEL
LIN {X 0,Y 401.479,Z 262.726,A -85,B 0,C 180,E1 19799.427,E2 19799.427} C_VEL
LIN {X 0,Y 401.472,Z 262.725,A -85,B 0,C 180,E1 19795.427,E2 19795.427} C_VEL
LIN {X 0,Y 401.473,Z 262.722,A -85,B 0,C 180,E1 19791.549,E2 19791.549} C_VEL
LIN {X 0,Y 401.462,Z 262.727,A -85,B 0,C 180,E1 19787.631,E2 19787.631} C_VEL
LIN {X 0,Y 401.441,Z 262.727,A -85,B 0,C 180,E1 19783.949,E2 19783.949} C_VEL
LIN {X 0,Y 401.439,Z 262.728,A -85,B 0,C 180,E1 19780.047,E2 19780.047} C_VEL
LIN {X 0,Y 401.437,Z 262.725,A -85,B 0,C 180,E1 19776.202,E2 19776.202} C_VEL
LIN {X 0,Y 401.44,Z 262.725,A -85,B 0,C 180,E1 19772.239,E2 19772.239} C_VEL
LIN {X 0,Y 401.449,Z 262.726,A -85,B 0,C 180,E1 19768.403,E2 19768.403} C_VEL
LIN {X 0,Y 401.5,Z 262.861,A -85,B 0,C 180,E1 19766.867,E2 19766.867} C_VEL
LIN {X 0,Y 402.779,Z 266.258,A -85,B 0,C 180,E1 19766.215,E2 19766.215} C_VEL
LIN {X 0,Y 404.001,Z 268.311,A -85,B 0,C 180,E1 19765.749,E2 19765.749} C_VEL
LIN {X 0,Y 410.38,Z 280.946,A -85,B 0,C 180,E1 19763.175,E2 19763.175} C_VEL
LIN {X 0,Y 416.605,Z 293.594,A -85,B 0,C 180,E1 19760.835,E2 19760.835} C_VEL
LIN {X 0,Y 430.303,Z 315.127,A -85,B 0,C 180,E1 19758.262,E2 19758.262} C_VEL
LIN {X 0,Y 441.597,Z 334.375,A -85,B 0,C 180,E1 19756.263,E2 19756.263} C_VEL
LIN {X 0,Y 442.678,Z 343.503,A -85,B 0,C 180,E1 19755.899,E2 19755.899} C_VEL
LIN {X 0,Y 434.716,Z 536.572,A -85,B 0,C 180,E1 19752.156,E2 19752.156} C_VEL
LIN {X 0,Y 432.096,Z 604.075,A -85,B 0,C 180,E1 19750.835,E2 19750.835} C_VEL
LIN {X 0,Y 430.236,Z 626.957,A -85,B 0,C 180,E1 19750.172,E2 19750.172} C_VEL
LIN {X 0,Y 428.057,Z 648.207,A -85,B 0,C 180,E1 19749.317,E2 19749.317} C_VEL
LIN {X 0,Y 425.563,Z 668.995,A -85,B 0,C 180,E1 19748.248,E2 19748.248} C_VEL
LIN {X 0,Y 422.652,Z 689.906,A -85,B 0,C 180,E1 19746.907,E2 19746.907} C_VEL
LIN {X 0,Y 419.558,Z 709.976,A -85,B 0,C 180,E1 19745.325,E2 19745.325} C_VEL
LIN {X 0,Y 416.437,Z 729.17,A -85,B 0,C 180,E1 19743.518,E2 19743.518} C_VEL
LIN {X 0,Y 413.428,Z 747.016,A -85,B 0,C 180,E1 19741.537,E2 19741.537} C_VEL
LIN {X 0,Y 410.501,Z 764.006,A -85,B 0,C 180,E1 19739.309,E2 19739.309} C_VEL
LIN {X 0,Y 407.927,Z 779.215,A -85,B 0,C 180,E1 19736.963,E2 19736.963} C_VEL
LIN {X 0,Y 405.561,Z 793.903,A -85,B 0,C 180,E1 19734.311,E2 19734.311} C_VEL
LIN {X 0,Y 403.707,Z 806.441,A -85,B 0,C 180,E1 19731.654,E2 19731.654} C_VEL
LIN {X 0,Y 402.24,Z 817.488,A -85,B 0,C 180,E1 19728.851,E2 19728.851} C_VEL
LIN {X 0,Y 401.168,Z 827.412,A -85,B 0,C 180,E1 19725.832,E2 19725.832} C_VEL
LIN {X 0,Y 400.528,Z 835.085,A -85,B 0,C 180,E1 19722.982,E2 19722.982} C_VEL
LIN {X 0,Y 400.18,Z 841.136,A -85,B 0,C 180,E1 19720.071,E2 19720.071} C_VEL
LIN {X 0,Y 400.042,Z 845.843,A -85,B 0,C 180,E1 19717.033,E2 19717.033} C_VEL
LIN {X 0,Y 399.999,Z 848.603,A -85,B 0,C 180,E1 19714.299,E2 19714.299} C_VEL
LIN {X 0,Y 400.004,Z 850.082,A -85,B 0,C 180,E1 19711.288,E2 19711.288} C_VEL
LIN {X 0,Y 400.007,Z 850.006,A -85,B 0,C 180,E1 19708.566,E2 19708.566} C_VEL
LIN {X 0,Y 400.014,Z 848.322,A -85,B 0,C 180,E1 19705.555,E2 19705.555} C_VEL
LIN {X 0,Y 400.059,Z 845.185,A -85,B 0,C 180,E1 19702.676,E2 19702.676} C_VEL
LIN {X 0,Y 400.218,Z 840.395,A -85,B 0,C 180,E1 19699.782,E2 19699.782} C_VEL
LIN {X 0,Y 400.591,Z 833.701,A -85,B 0,C 180,E1 19696.763,E2 19696.763} C_VEL
LIN {X 0,Y 401.234,Z 825.673,A -85,B 0,C 180,E1 19693.941,E2 19693.941} C_VEL
LIN {X 0,Y 402.209,Z 815.95,A -85,B 0,C 180,E1 19691.144,E2 19691.144} C_VEL
LIN {X 0,Y 403.532,Z 804.978,A -85,B 0,C 180,E1 19688.486,E2 19688.486} C_VEL
LIN {X 0,Y 405.272,Z 791.795,A -85,B 0,C 180,E1 19685.823,E2 19685.823} C_VEL
LIN {X 0,Y 407.346,Z 777.199,A -85,B 0,C 180,E1 19683.307,E2 19683.307} C_VEL
LIN {X 0,Y 409.718,Z 761.155,A -85,B 0,C 180,E1 19680.945,E2 19680.945} C_VEL
LIN {X 0,Y 412.271,Z 744.132,A -85,B 0,C 180,E1 19678.815,E2 19678.815} C_VEL
LIN {X 0,Y 415,Z 725.63,A -85,B 0,C 180,E1 19676.844,E2 19676.844} C_VEL
LIN {X 0,Y 417.838,Z 705.646,A -85,B 0,C 180,E1 19675.033,E2 19675.033} C_VEL
LIN {X 0,Y 420.692,Z 684.721,A -85,B 0,C 180,E1 19673.45,E2 19673.45} C_VEL
LIN {X 0,Y 423.352,Z 663.107,A -85,B 0,C 180,E1 19672.115,E2 19672.115} C_VEL
LIN {X 0,Y 425.827,Z 640.899,A -85,B 0,C 180,E1 19671.002,E2 19671.002} C_VEL
LIN {X 0,Y 428.197,Z 617.198,A -85,B 0,C 180,E1 19670.091,E2 19670.091} C_VEL
LIN {X 0,Y 430.038,Z 593.489,A -85,B 0,C 180,E1 19669.414,E2 19669.414} C_VEL
LIN {X 0,Y 435.149,Z 487.159,A -85,B 0,C 180,E1 19667.142,E2 19667.142} C_VEL
LIN {X 0,Y 440.851,Z 402.778,A -85,B 0,C 180,E1 19665.181,E2 19665.181} C_VEL
LIN {X 0,Y 446,Z 342.272,A -85,B 0,C 180,E1 19663.67,E2 19663.67} C_VEL
LIN {X 0,Y 445.61,Z 333.095,A -85,B 0,C 180,E1 19663.164,E2 19663.164} C_VEL
LIN {X 0,Y 442.335,Z 322.733,A -85,B 0,C 180,E1 19661.8,E2 19661.8} C_VEL
LIN {X 0,Y 440.188,Z 316.332,A -85,B 0,C 180,E1 19660.686,E2 19660.686} C_VEL
LIN {X 0,Y 438.38,Z 310.861,A -85,B 0,C 180,E1 19659.394,E2 19659.394} C_VEL
LIN {X 0,Y 437.568,Z 307.967,A -85,B 0,C 180,E1 19658.471,E2 19658.471} C_VEL
LIN {X 0,Y 437.244,Z 305.955,A -85,B 0,C 180,E1 19657.631,E2 19657.631} C_VEL
LIN {X 0,Y 437.516,Z 304.38,A -85,B 0,C 180,E1 19655.968,E2 19655.968} C_VEL
LIN {X 0,Y 437.974,Z 304.405,A -85,B 0,C 180,E1 19655.362,E2 19655.362} C_VEL
LIN {X 0,Y 439.92,Z 308.281,A -85,B 0,C 180,E1 19653.612,E2 19653.612} C_VEL
LIN {X 0,Y 442.139,Z 312.791,A -85,B 0,C 180,E1 19652.41,E2 19652.41} C_VEL
LIN {X 0,Y 445.166,Z 318.87,A -85,B 0,C 180,E1 19651.189,E2 19651.189} C_VEL
LIN {X 0,Y 447.026,Z 323.367,A -85,B 0,C 180,E1 19650.522,E2 19650.522} C_VEL
LIN {X 0,Y 439.949,Z 401.116,A -85,B 0,C 180,E1 19648.605,E2 19648.605} C_VEL
LIN {X 0,Y 434.68,Z 479.808,A -85,B 0,C 180,E1 19646.79,E2 19646.79} C_VEL
LIN {X 0,Y 431.24,Z 547.238,A -85,B 0,C 180,E1 19645.3,E2 19645.3} C_VEL
LIN {X 0,Y 429.7,Z 569.759,A -85,B 0,C 180,E1 19644.549,E2 19644.549} C_VEL
LIN {X 0,Y 427.751,Z 590.768,A -85,B 0,C 180,E1 19643.609,E2 19643.609} C_VEL
LIN {X 0,Y 425.438,Z 611.15,A -85,B 0,C 180,E1 19642.453,E2 19642.453} C_VEL
LIN {X 0,Y 422.933,Z 630.236,A -85,B 0,C 180,E1 19641.134,E2 19641.134} C_VEL
LIN {X 0,Y 420.02,Z 649.997,A -85,B 0,C 180,E1 19639.469,E2 19639.469} C_VEL
LIN {X 0,Y 417.134,Z 667.19,A -85,B 0,C 180,E1 19637.724,E2 19637.724} C_VEL
LIN {X 0,Y 414.146,Z 684.171,A -85,B 0,C 180,E1 19635.689,E2 19635.689} C_VEL
LIN {X 0,Y 411.47,Z 698.793,A -85,B 0,C 180,E1 19633.635,E2 19633.635} C_VEL
LIN {X 0,Y 408.814,Z 712.917,A -85,B 0,C 180,E1 19631.285,E2 19631.285} C_VEL
LIN {X 0,Y 406.442,Z 725.682,A -85,B 0,C 180,E1 19628.775,E2 19628.775} C_VEL
LIN {X 0,Y 404.429,Z 737.183,A -85,B 0,C 180,E1 19626.104,E2 19626.104} C_VEL
LIN {X 0,Y 402.801,Z 747.273,A -85,B 0,C 180,E1 19623.275,E2 19623.275} C_VEL
LIN {X 0,Y 401.627,Z 755.537,A -85,B 0,C 180,E1 19620.43,E2 19620.43} C_VEL
LIN {X 0,Y 400.815,Z 762.563,A -85,B 0,C 180,E1 19617.428,E2 19617.428} C_VEL
LIN {X 0,Y 400.362,Z 767.952,A -85,B 0,C 180,E1 19614.413,E2 19614.413} C_VEL
LIN {X 0,Y 400.12,Z 771.733,A -85,B 0,C 180,E1 19611.379,E2 19611.379} C_VEL
LIN {X 0,Y 400.033,Z 774.1,A -85,B 0,C 180,E1 19608.322,E2 19608.322} C_VEL
LIN {X 0,Y 400.023,Z 774.924,A -85,B 0,C 180,E1 19605.312,E2 19605.312} C_VEL
LIN {X 0,Y 400.016,Z 774.258,A -85,B 0,C 180,E1 19602.239,E2 19602.239} C_VEL
LIN {X 0,Y 400.076,Z 772.161,A -85,B 0,C 180,E1 19599.18,E2 19599.18} C_VEL
LIN {X 0,Y 400.235,Z 768.422,A -85,B 0,C 180,E1 19596.113,E2 19596.113} C_VEL
LIN {X 0,Y 400.641,Z 762.982,A -85,B 0,C 180,E1 19592.989,E2 19592.989} C_VEL
LIN {X 0,Y 401.367,Z 756.057,A -85,B 0,C 180,E1 19589.956,E2 19589.956} C_VEL
LIN {X 0,Y 402.454,Z 747.644,A -85,B 0,C 180,E1 19587.041,E2 19587.041} C_VEL
LIN {X 0,Y 403.946,Z 737.844,A -85,B 0,C 180,E1 19584.26,E2 19584.26} C_VEL
LIN {X 0,Y 405.961,Z 726.046,A -85,B 0,C 180,E1 19581.459,E2 19581.459} C_VEL
LIN {X 0,Y 408.39,Z 712.742,A -85,B 0,C 180,E1 19578.811,E2 19578.811} C_VEL
LIN {X 0,Y 411.035,Z 698.375,A -85,B 0,C 180,E1 19576.413,E2 19576.413} C_VEL
LIN {X 0,Y 414.121,Z 681.723,A -85,B 0,C 180,E1 19574.056,E2 19574.056} C_VEL
LIN {X 0,Y 417.199,Z 664.721,A -85,B 0,C 180,E1 19572.021,E2 19572.021} C_VEL
LIN {X 0,Y 420.261,Z 646.786,A -85,B 0,C 180,E1 19570.213,E2 19570.213} C_VEL
LIN {X 0,Y 423.139,Z 628.256,A -85,B 0,C 180,E1 19568.646,E2 19568.646} C_VEL
LIN {X 0,Y 425.961,Z 608.409,A -85,B 0,C 180,E1 19567.248,E2 19567.248} C_VEL
LIN {X 0,Y 428.427,Z 588.34,A -85,B 0,C 180,E1 19566.097,E2 19566.097} C_VEL
LIN {X 0,Y 430.544,Z 566.681,A -85,B 0,C 180,E1 19565.124,E2 19565.124} C_VEL
LIN {X 0,Y 432.307,Z 543.741,A -85,B 0,C 180,E1 19564.359,E2 19564.359} C_VEL
LIN {X 0,Y 433.533,Z 520.135,A -85,B 0,C 180,E1 19563.823,E2 19563.823} C_VEL
LIN {X 0,Y 441.352,Z 323.693,A -85,B 0,C 180,E1 19560.052,E2 19560.052} C_VEL
LIN {X 0,Y 441.255,Z 321.216,A -85,B 0,C 180,E1 19559.977,E2 19559.977} C_VEL
LIN {X 0,Y 428.652,Z 302.005,A -85,B 0,C 180,E1 19557.847,E2 19557.847} C_VEL
LIN {X 0,Y 415.591,Z 283.355,A -85,B 0,C 180,E1 19555.472,E2 19555.472} C_VEL
LIN {X 0,Y 408.329,Z 273.345,A -85,B 0,C 180,E1 19554.069,E2 19554.069} C_VEL
LIN {X 0,Y 405.59,Z 269.543,A -85,B 0,C 180,E1 19553.52,E2 19553.52} C_VEL
LIN {X 0,Y 404.664,Z 268.147,A -85,B 0,C 180,E1 19553.326,E2 19553.326} C_VEL
LIN {X 0,Y 404.457,Z 267.986,A -85,B 0,C 180,E1 19553.288,E2 19553.288} C_VEL
LIN {X 0,Y 399.544,Z 265.247,A -85,B 0,C 180,E1 19552.374,E2 19552.374} C_VEL
LIN {X 0,Y 395.561,Z 264.07,A -85,B 0,C 180,E1 19551.442,E2 19551.442} C_VEL
LIN {X 0,Y 393.716,Z 263.735,A -85,B 0,C 180,E1 19550.609,E2 19550.609} C_VEL
LIN {X 0,Y 393.53,Z 263.714,A -85,B 0,C 180,E1 19550.281,E2 19550.281} C_VEL
LIN {X 0,Y 393.533,Z 263.71,A -85,B 0,C 180,E1 19546.382,E2 19546.382} C_VEL
LIN {X 0,Y 393.54,Z 263.716,A -85,B 0,C 180,E1 19542.473,E2 19542.473} C_VEL
LIN {X 0,Y 393.542,Z 263.707,A -85,B 0,C 180,E1 19538.475,E2 19538.475} C_VEL
LIN {X 0,Y 393.554,Z 263.706,A -85,B 0,C 180,E1 19534.665,E2 19534.665} C_VEL
LIN {X 0,Y 393.566,Z 263.709,A -85,B 0,C 180,E1 19530.729,E2 19530.729} C_VEL
LIN {X 0,Y 393.556,Z 263.707,A -85,B 0,C 180,E1 19526.745,E2 19526.745} C_VEL
LIN {X 0,Y 393.571,Z 263.702,A -85,B 0,C 180,E1 19522.704,E2 19522.704} C_VEL
LIN {X 0,Y 393.554,Z 263.703,A -85,B 0,C 180,E1 19518.698,E2 19518.698} C_VEL
LIN {X 0,Y 393.56,Z 263.703,A -85,B 0,C 180,E1 19514.681,E2 19514.681} C_VEL
LIN {X 0,Y 393.55,Z 263.706,A -85,B 0,C 180,E1 19510.716,E2 19510.716} C_VEL
LIN {X 0,Y 393.538,Z 263.71,A -85,B 0,C 180,E1 19506.81,E2 19506.81} C_VEL
LIN {X 0,Y 393.525,Z 263.715,A -85,B 0,C 180,E1 19502.95,E2 19502.95} C_VEL
LIN {X 0,Y 393.514,Z 263.717,A -85,B 0,C 180,E1 19499.122,E2 19499.122} C_VEL
LIN {X 0,Y 393.508,Z 263.719,A -85,B 0,C 180,E1 19495.15,E2 19495.15} C_VEL
LIN {X 0,Y 393.506,Z 263.72,A -85,B 0,C 180,E1 19491.261,E2 19491.261} C_VEL
LIN {X 0,Y 393.505,Z 263.719,A -85,B 0,C 180,E1 19487.245,E2 19487.245} C_VEL
LIN {X 0,Y 393.505,Z 263.715,A -85,B 0,C 180,E1 19483.314,E2 19483.314} C_VEL
LIN {X 0,Y 393.506,Z 263.71,A -85,B 0,C 180,E1 19479.43,E2 19479.43} C_VEL
LIN {X 0,Y 393.518,Z 263.71,A -85,B 0,C 180,E1 19475.577,E2 19475.577} C_VEL
LIN {X 0,Y 393.526,Z 263.714,A -85,B 0,C 180,E1 19471.666,E2 19471.666} C_VEL
LIN {X 0,Y 393.549,Z 263.716,A -85,B 0,C 180,E1 19467.859,E2 19467.859} C_VEL
LIN {X 0,Y 393.542,Z 263.714,A -85,B 0,C 180,E1 19463.824,E2 19463.824} C_VEL
LIN {X 0,Y 393.536,Z 263.715,A -85,B 0,C 180,E1 19459.902,E2 19459.902} C_VEL
LIN {X 0,Y 393.53,Z 263.717,A -85,B 0,C 180,E1 19455.924,E2 19455.924} C_VEL
LIN {X 0,Y 393.516,Z 263.719,A -85,B 0,C 180,E1 19451.991,E2 19451.991} C_VEL
LIN {X 0,Y 393.508,Z 263.719,A -85,B 0,C 180,E1 19448.031,E2 19448.031} C_VEL
LIN {X 0,Y 393.493,Z 263.718,A -85,B 0,C 180,E1 19444.224,E2 19444.224} C_VEL
LIN {X 0,Y 393.489,Z 263.713,A -85,B 0,C 180,E1 19440.289,E2 19440.289} C_VEL
LIN {X 0,Y 393.489,Z 263.719,A -85,B 0,C 180,E1 19436.356,E2 19436.356} C_VEL
LIN {X 0,Y 393.491,Z 263.718,A -85,B 0,C 180,E1 19432.405,E2 19432.405} C_VEL
LIN {X 0,Y 393.493,Z 263.716,A -85,B 0,C 180,E1 19428.418,E2 19428.418} C_VEL
LIN {X 0,Y 393.498,Z 263.717,A -85,B 0,C 180,E1 19424.524,E2 19424.524} C_VEL
LIN {X 0,Y 393.511,Z 263.713,A -85,B 0,C 180,E1 19420.711,E2 19420.711} C_VEL
LIN {X 0,Y 393.522,Z 263.71,A -85,B 0,C 180,E1 19416.806,E2 19416.806} C_VEL
LIN {X 0,Y 393.54,Z 263.711,A -85,B 0,C 180,E1 19412.948,E2 19412.948} C_VEL
LIN {X 0,Y 393.547,Z 263.711,A -85,B 0,C 180,E1 19408.951,E2 19408.951} C_VEL
LIN {X 0,Y 393.513,Z 263.795,A -85,B 0,C 180,E1 19408.165,E2 19408.165} C_VEL
LIN {X 0,Y 394.753,Z 267.091,A -85,B 0,C 180,E1 19407.502,E2 19407.502} C_VEL
LIN {X 0,Y 395.873,Z 268.557,A -85,B 0,C 180,E1 19407.109,E2 19407.109} C_VEL
LIN {X 0,Y 397.788,Z 272.584,A -85,B 0,C 180,E1 19406.254,E2 19406.254} C_VEL
LIN {X 0,Y 404.683,Z 286.332,A -85,B 0,C 180,E1 19403.413,E2 19403.413} C_VEL
LIN {X 0,Y 408.016,Z 292.96,A -85,B 0,C 180,E1 19402.174,E2 19402.174} C_VEL
LIN {X 0,Y 422.264,Z 315.111,A -85,B 0,C 180,E1 19399.37,E2 19399.37} C_VEL
LIN {X 0,Y 434.858,Z 336.17,A -85,B 0,C 180,E1 19397.087,E2 19397.087} C_VEL
LIN {X 0,Y 436.232,Z 339.083,A -85,B 0,C 180,E1 19396.828,E2 19396.828} C_VEL
LIN {X 0,Y 436.814,Z 345.281,A -85,B 0,C 180,E1 19396.589,E2 19396.589} C_VEL
LIN {X 0,Y 428.455,Z 536.882,A -85,B 0,C 180,E1 19392.816,E2 19392.816} C_VEL
LIN {X 0,Y 425.688,Z 603.571,A -85,B 0,C 180,E1 19391.484,E2 19391.484} C_VEL
LIN {X 0,Y 423.74,Z 626.465,A -85,B 0,C 180,E1 19390.812,E2 19390.812} C_VEL
LIN {X 0,Y 421.401,Z 648.198,A -85,B 0,C 180,E1 19389.925,E2 19389.925} C_VEL
LIN {X 0,Y 418.561,Z 670.525,A -85,B 0,C 180,E1 19388.743,E2 19388.743} C_VEL
LIN {X 0,Y 415.597,Z 690.89,A -85,B 0,C 180,E1 19387.405,E2 19387.405} C_VEL
LIN {X 0,Y 412.404,Z 710.707,A -85,B 0,C 180,E1 19385.81,E2 19385.81} C_VEL
LIN {X 0,Y 409.224,Z 729.265,A -85,B 0,C 180,E1 19384.02,E2 19384.02} C_VEL
LIN {X 0,Y 406.004,Z 747.319,A -85,B 0,C 180,E1 19381.968,E2 19381.968} C_VEL
LIN {X 0,Y 402.987,Z 764.062,A -85,B 0,C 180,E1 19379.726,E2 19379.726} C_VEL
LIN {X 0,Y 400.305,Z 779.063,A -85,B 0,C 180,E1 19377.358,E2 19377.358} C_VEL
LIN {X 0,Y 397.819,Z 793.709,A -85,B 0,C 180,E1 19374.657,E2 19374.657} C_VEL
LIN {X 0,Y 395.87,Z 806.197,A -85,B 0,C 180,E1 19371.949,E2 19371.949} C_VEL
LIN {X 0,Y 394.334,Z 817.192,A -85,B 0,C 180,E1 19369.09,E2 19369.09} C_VEL
LIN {X 0,Y 393.211,Z 827.026,A -85,B 0,C 180,E1 19366.015,E2 19366.015} C_VEL
LIN {X 0,Y 392.548,Z 834.65,A -85,B 0,C 180,E1 19363.101,E2 19363.101} C_VEL
LIN {X 0,Y 392.195,Z 840.65,A -85,B 0,C 180,E1 19360.13,E2 19360.13} C_VEL
LIN {X 0,Y 392.061,Z 845.277,A -85,B 0,C 180,E1 19357.03,E2 19357.03} C_VEL
LIN {X 0,Y 392.025,Z 847.982,A -85,B 0,C 180,E1 19354.24,E2 19354.24} C_VEL
LIN {X 0,Y 392.04,Z 849.368,A -85,B 0,C 180,E1 19351.168,E2 19351.168} C_VEL
LIN {X 0,Y 392.04,Z 849.21,A -85,B 0,C 180,E1 19348.391,E2 19348.391} C_VEL
LIN {X 0,Y 392.049,Z 847.403,A -85,B 0,C 180,E1 19345.317,E2 19345.317} C_VEL
LIN {X 0,Y 392.083,Z 844.158,A -85,B 0,C 180,E1 19342.378,E2 19342.378} C_VEL
LIN {X 0,Y 392.27,Z 839.204,A -85,B 0,C 180,E1 19339.424,E2 19339.424} C_VEL
LIN {X 0,Y 392.652,Z 832.62,A -85,B 0,C 180,E1 19336.45,E2 19336.45} C_VEL
LIN {X 0,Y 393.328,Z 824.627,A -85,B 0,C 180,E1 19333.609,E2 19333.609} C_VEL
LIN {X 0,Y 394.433,Z 814.244,A -85,B 0,C 180,E1 19330.604,E2 19330.604} C_VEL
LIN {X 0,Y 395.935,Z 802.304,A -85,B 0,C 180,E1 19327.74,E2 19327.74} C_VEL
LIN {X 0,Y 397.736,Z 789.606,A -85,B 0,C 180,E1 19325.165,E2 19325.165} C_VEL
LIN {X 0,Y 399.967,Z 774.753,A -85,B 0,C 180,E1 19322.613,E2 19322.613} C_VEL
LIN {X 0,Y 402.528,Z 758.423,A -85,B 0,C 180,E1 19320.211,E2 19320.211} C_VEL
LIN {X 0,Y 405.345,Z 740.525,A -85,B 0,C 180,E1 19317.971,E2 19317.971} C_VEL
LIN {X 0,Y 408.169,Z 722.268,A -85,B 0,C 180,E1 19316.046,E2 19316.046} C_VEL
LIN {X 0,Y 411.203,Z 701.824,A -85,B 0,C 180,E1 19314.211,E2 19314.211} C_VEL
LIN {X 0,Y 414.238,Z 680.512,A -85,B 0,C 180,E1 19312.622,E2 19312.622} C_VEL
LIN {X 0,Y 417.11,Z 658.455,A -85,B 0,C 180,E1 19311.269,E2 19311.269} C_VEL
LIN {X 0,Y 419.801,Z 635.526,A -85,B 0,C 180,E1 19310.156,E2 19310.156} C_VEL
LIN {X 0,Y 422.221,Z 611.769,A -85,B 0,C 180,E1 19309.273,E2 19309.273} C_VEL
LIN {X 0,Y 424.117,Z 586.728,A -85,B 0,C 180,E1 19308.59,E2 19308.59} C_VEL
LIN {X 0,Y 429.205,Z 492.373,A -85,B 0,C 180,E1 19306.502,E2 19306.502} C_VEL
LIN {X 0,Y 435.292,Z 411.035,A -85,B 0,C 180,E1 19304.549,E2 19304.549} C_VEL
LIN {X 0,Y 441.673,Z 344.151,A -85,B 0,C 180,E1 19302.827,E2 19302.827} C_VEL
LIN {X 0,Y 441.511,Z 337.196,A -85,B 0,C 180,E1 19302.423,E2 19302.423} C_VEL
LIN {X 0,Y 438.976,Z 328.09,A -85,B 0,C 180,E1 19301.147,E2 19301.147} C_VEL
LIN {X 0,Y 437.401,Z 322.587,A -85,B 0,C 180,E1 19300.139,E2 19300.139} C_VEL
LIN {X 0,Y 436.074,Z 317.512,A -85,B 0,C 180,E1 19298.88,E2 19298.88} C_VEL
LIN {X 0,Y 435.508,Z 313.721,A -85,B 0,C 180,E1 19297.516,E2 19297.516} C_VEL
LIN {X 0,Y 435.946,Z 312.15,A -85,B 0,C 180,E1 19295.794,E2 19295.794} C_VEL
LIN {X 0,Y 436.201,Z 312.424,A -85,B 0,C 180,E1 19295.402,E2 19295.402} C_VEL
LIN {X 0,Y 437.715,Z 315.778,A -85,B 0,C 180,E1 19293.875,E2 19293.875} C_VEL
LIN {X 0,Y 439.747,Z 320.346,A -85,B 0,C 180,E1 19292.65,E2 19292.65} C_VEL
LIN {X 0,Y 442.748,Z 327.134,A -85,B 0,C 180,E1 19291.338,E2 19291.338} C_VEL
LIN {X 0,Y 434.696,Z 406.415,A -85,B 0,C 180,E1 19289.318,E2 19289.318} C_VEL
LIN {X 0,Y 429.087,Z 480.49,A -85,B 0,C 180,E1 19287.543,E2 19287.543} C_VEL
LIN {X 0,Y 425.132,Z 548.943,A -85,B 0,C 180,E1 19285.966,E2 19285.966} C_VEL
LIN {X 0,Y 423.449,Z 571.672,A -85,B 0,C 180,E1 19285.181,E2 19285.181} C_VEL
LIN {X 0,Y 421.396,Z 592.227,A -85,B 0,C 180,E1 19284.236,E2 19284.236} C_VEL
LIN {X 0,Y 418.922,Z 612.791,A -85,B 0,C 180,E1 19283.045,E2 19283.045} C_VEL
LIN {X 0,Y 416.158,Z 632.492,A -85,B 0,C 180,E1 19281.643,E2 19281.643} C_VEL
LIN {X 0,Y 413.233,Z 651.326,A -85,B 0,C 180,E1 19280.023,E2 19280.023} C_VEL
LIN {X 0,Y 409.987,Z 669.679,A -85,B 0,C 180,E1 19278.117,E2 19278.117} C_VEL
LIN {X 0,Y 406.962,Z 685.862,A -85,B 0,C 180,E1 19276.12,E2 19276.12} C_VEL
LIN {X 0,Y 403.971,Z 701.225,A -85,B 0,C 180,E1 19273.893,E2 19273.893} C_VEL
LIN {X 0,Y 401.221,Z 715.178,A -85,B 0,C 180,E1 19271.501,E2 19271.501} C_VEL
LIN {X 0,Y 398.749,Z 727.723,A -85,B 0,C 180,E1 19268.945,E2 19268.945} C_VEL
LIN {X 0,Y 396.541,Z 739.517,A -85,B 0,C 180,E1 19266.081,E2 19266.081} C_VEL
LIN {X 0,Y 394.876,Z 749.393,A -85,B 0,C 180,E1 19263.195,E2 19263.195} C_VEL
LIN {X 0,Y 393.681,Z 757.439,A -85,B 0,C 180,E1 19260.293,E2 19260.293} C_VEL
LIN {X 0,Y 392.849,Z 764.186,A -85,B 0,C 180,E1 19257.23,E2 19257.23} C_VEL
LIN {X 0,Y 392.393,Z 769.372,A -85,B 0,C 180,E1 19254.152,E2 19254.152} C_VEL
LIN {X 0,Y 392.159,Z 772.811,A -85,B 0,C 180,E1 19251.203,E2 19251.203} C_VEL
LIN {X 0,Y 392.063,Z 774.984,A -85,B 0,C 180,E1 19248.081,E2 19248.081} C_VEL
LIN {X 0,Y 392.06,Z 775.7,A -85,B 0,C 180,E1 19245.076,E2 19245.076} C_VEL
LIN {X 0,Y 392.053,Z 774.904,A -85,B 0,C 180,E1 19242.028,E2 19242.028} C_VEL
LIN {X 0,Y 392.12,Z 772.707,A -85,B 0,C 180,E1 19238.931,E2 19238.931} C_VEL
LIN {X 0,Y 392.302,Z 769.096,A -85,B 0,C 180,E1 19235.937,E2 19235.937} C_VEL
LIN {X 0,Y 392.75,Z 763.576,A -85,B 0,C 180,E1 19232.729,E2 19232.729} C_VEL
LIN {X 0,Y 393.544,Z 756.581,A -85,B 0,C 180,E1 19229.633,E2 19229.633} C_VEL
LIN {X 0,Y 394.726,Z 748.107,A -85,B 0,C 180,E1 19226.659,E2 19226.659} C_VEL
LIN {X 0,Y 396.328,Z 738.218,A -85,B 0,C 180,E1 19223.823,E2 19223.823} C_VEL
LIN {X 0,Y 398.382,Z 726.849,A -85,B 0,C 180,E1 19221.082,E2 19221.082} C_VEL
LIN {X 0,Y 400.884,Z 713.784,A -85,B 0,C 180,E1 19218.439,E2 19218.439} C_VEL
LIN {X 0,Y 403.666,Z 699.429,A -85,B 0,C 180,E1 19215.994,E2 19215.994} C_VEL
LIN {X 0,Y 406.77,Z 683.511,A -85,B 0,C 180,E1 19213.688,E2 19213.688} C_VEL
LIN {X 0,Y 409.96,Z 666.786,A -85,B 0,C 180,E1 19211.628,E2 19211.628} C_VEL
LIN {X 0,Y 413.126,Z 648.996,A -85,B 0,C 180,E1 19209.792,E2 19209.792} C_VEL
LIN {X 0,Y 416.269,Z 629.69,A -85,B 0,C 180,E1 19208.12,E2 19208.12} C_VEL
LIN {X 0,Y 419.237,Z 609.644,A -85,B 0,C 180,E1 19206.684,E2 19206.684} C_VEL
LIN {X 0,Y 421.823,Z 589.325,A -85,B 0,C 180,E1 19205.503,E2 19205.503} C_VEL
LIN {X 0,Y 424.029,Z 567.825,A -85,B 0,C 180,E1 19204.519,E2 19204.519} C_VEL
LIN {X 0,Y 425.896,Z 544.682,A -85,B 0,C 180,E1 19203.73,E2 19203.73} C_VEL
LIN {X 0,Y 427.17,Z 521.731,A -85,B 0,C 180,E1 19203.195,E2 19203.195} C_VEL
LIN {X 0,Y 434.771,Z 340.157,A -85,B 0,C 180,E1 19199.651,E2 19199.651} C_VEL
LIN {X 0,Y 435.357,Z 324.759,A -85,B 0,C 180,E1 19199.326,E2 19199.326} C_VEL
LIN {X 0,Y 421.511,Z 303.804,A -85,B 0,C 180,E1 19196.923,E2 19196.923} C_VEL
LIN {X 0,Y 407.773,Z 284.368,A -85,B 0,C 180,E1 19194.328,E2 19194.328} C_VEL
LIN {X 0,Y 403.783,Z 279.03,A -85,B 0,C 180,E1 19193.535,E2 19193.535} C_VEL
LIN {X 0,Y 400.492,Z 274.336,A -85,B 0,C 180,E1 19192.845,E2 19192.845} C_VEL
LIN {X 0,Y 397.723,Z 270.429,A -85,B 0,C 180,E1 19192.252,E2 19192.252} C_VEL
LIN {X 0,Y 396.784,Z 269.214,A -85,B 0,C 180,E1 19192.054,E2 19192.054} C_VEL
LIN {X 0,Y 394.38,Z 266.402,A -85,B 0,C 180,E1 19191.55,E2 19191.55} C_VEL
LIN {X 0,Y 393.563,Z 263.707,A -85,B 0,C 180,E1 19191.304,E2 19191.304} C_VEL
LIN {X 0,Y 393.53,Z 263.714,A -85,B 0,C 180,E1 19190.281,E2 19190.281} C_VEL
LIN {X 0,Y 392.519,Z 263.846,A -85,B 0,C 180,E1 19189.159,E2 19189.159} C_VEL
LIN {X 0,Y 386.032,Z 264.646,A -85,B 0,C 180,E1 19185.913,E2 19185.913} C_VEL
LIN {X 0,Y 385.625,Z 264.701,A -85,B 0,C 180,E1 19185.168,E2 19185.168} C_VEL
LIN {X 0,Y 385.613,Z 264.695,A -85,B 0,C 180,E1 19181.215,E2 19181.215} C_VEL
LIN {X 0,Y 385.615,Z 264.699,A -85,B 0,C 180,E1 19177.151,E2 19177.151} C_VEL
LIN {X 0,Y 385.608,Z 264.697,A -85,B 0,C 180,E1 19173.123,E2 19173.123} C_VEL
LIN {X 0,Y 385.597,Z 264.692,A -85,B 0,C 180,E1 19169.259,E2 19169.259} C_VEL
LIN {X 0,Y 385.593,Z 264.689,A -85,B 0,C 180,E1 19165.242,E2 19165.242} C_VEL
LIN {X 0,Y 385.585,Z 264.695,A -85,B 0,C 180,E1 19161.352,E2 19161.352} C_VEL
LIN {X 0,Y 385.58,Z 264.698,A -85,B 0,C 180,E1 19157.42,E2 19157.42} C_VEL
LIN {X 0,Y 385.578,Z 264.7,A -85,B 0,C 180,E1 19153.428,E2 19153.428} C_VEL
LIN {X 0,Y 385.575,Z 264.7,A -85,B 0,C 180,E1 19149.402,E2 19149.402} C_VEL
LIN {X 0,Y 385.573,Z 264.699,A -85,B 0,C 180,E1 19145.488,E2 19145.488} C_VEL
LIN {X 0,Y 385.572,Z 264.698,A -85,B 0,C 180,E1 19141.503,E2 19141.503} C_VEL
LIN {X 0,Y 385.571,Z 264.696,A -85,B 0,C 180,E1 19137.537,E2 19137.537} C_VEL
LIN {X 0,Y 385.574,Z 264.699,A -85,B 0,C 180,E1 19133.573,E2 19133.573} C_VEL
LIN {X 0,Y 385.58,Z 264.704,A -85,B 0,C 180,E1 19129.67,E2 19129.67} C_VEL
LIN {X 0,Y 385.588,Z 264.708,A -85,B 0,C 180,E1 19125.773,E2 19125.773} C_VEL
LIN {X 0,Y 385.592,Z 264.71,A -85,B 0,C 180,E1 19121.787,E2 19121.787} C_VEL
LIN {X 0,Y 385.605,Z 264.703,A -85,B 0,C 180,E1 19117.914,E2 19117.914} C_VEL
LIN {X 0,Y 385.601,Z 264.697,A -85,B 0,C 180,E1 19113.879,E2 19113.879} C_VEL
LIN {X 0,Y 385.608,Z 264.693,A -85,B 0,C 180,E1 19109.854,E2 19109.854} C_VEL
LIN {X 0,Y 385.598,Z 264.693,A -85,B 0,C 180,E1 19105.822,E2 19105.822} C_VEL
LIN {X 0,Y 385.607,Z 264.696,A -85,B 0,C 180,E1 19101.762,E2 19101.762} C_VEL
LIN {X 0,Y 385.595,Z 264.698,A -85,B 0,C 180,E1 19097.658,E2 19097.658} C_VEL
LIN {X 0,Y 385.6,Z 264.698,A -85,B 0,C 180,E1 19093.646,E2 19093.646} C_VEL
LIN {X 0,Y 385.59,Z 264.703,A -85,B 0,C 180,E1 19089.551,E2 19089.551} C_VEL
LIN {X 0,Y 385.593,Z 264.706,A -85,B 0,C 180,E1 19085.653,E2 19085.653} C_VEL
LIN {X 0,Y 385.592,Z 264.703,A -85,B 0,C 180,E1 19081.484,E2 19081.484} C_VEL
LIN {X 0,Y 385.59,Z 264.7,A -85,B 0,C 180,E1 19077.472,E2 19077.472} C_VEL
LIN {X 0,Y 385.604,Z 264.702,A -85,B 0,C 180,E1 19073.447,E2 19073.447} C_VEL
LIN {X 0,Y 385.595,Z 264.701,A -85,B 0,C 180,E1 19069.333,E2 19069.333} C_VEL
LIN {X 0,Y 385.611,Z 264.7,A -85,B 0,C 180,E1 19065.266,E2 19065.266} C_VEL
LIN {X 0,Y 385.6,Z 264.697,A -85,B 0,C 180,E1 19061.157,E2 19061.157} C_VEL
LIN {X 0,Y 385.609,Z 264.697,A -85,B 0,C 180,E1 19057.11,E2 19057.11} C_VEL
LIN {X 0,Y 385.605,Z 264.699,A -85,B 0,C 180,E1 19053.013,E2 19053.013} C_VEL
LIN {X 0,Y 385.605,Z 264.886,A -85,B 0,C 180,E1 19049.488,E2 19049.488} C_VEL
LIN {X 0,Y 387.069,Z 268.433,A -85,B 0,C 180,E1 19048.719,E2 19048.719} C_VEL
LIN {X 0,Y 388.099,Z 270.167,A -85,B 0,C 180,E1 19048.292,E2 19048.292} C_VEL
LIN {X 0,Y 390.989,Z 275.979,A -85,B 0,C 180,E1 19046.995,E2 19046.995} C_VEL
LIN {X 0,Y 395.363,Z 284.533,A -85,B 0,C 180,E1 19045.141,E2 19045.141} C_VEL
LIN {X 0,Y 399.231,Z 292.056,A -85,B 0,C 180,E1 19043.633,E2 19043.633} C_VEL
LIN {X 0,Y 412.036,Z 311.588,A -85,B 0,C 180,E1 19040.97,E2 19040.97} C_VEL
LIN {X 0,Y 424.592,Z 331.991,A -85,B 0,C 180,E1 19038.568,E2 19038.568} C_VEL
LIN {X 0,Y 430.776,Z 342.946,A -85,B 0,C 180,E1 19037.444,E2 19037.444} C_VEL
LIN {X 0,Y 431.028,Z 347.166,A -85,B 0,C 180,E1 19037.297,E2 19037.297} C_VEL
LIN {X 0,Y 422.126,Z 539.364,A -85,B 0,C 180,E1 19033.447,E2 19033.447} C_VEL
LIN {X 0,Y 419.334,Z 603.075,A -85,B 0,C 180,E1 19032.152,E2 19032.152} C_VEL
LIN {X 0,Y 417.315,Z 625.846,A -85,B 0,C 180,E1 19031.475,E2 19031.475} C_VEL
LIN {X 0,Y 414.888,Z 647.344,A -85,B 0,C 180,E1 19030.591,E2 19030.591} C_VEL
LIN {X 0,Y 411.933,Z 669.707,A -85,B 0,C 180,E1 19029.397,E2 19029.397} C_VEL
LIN {X 0,Y 408.834,Z 690.089,A -85,B 0,C 180,E1 19028.044,E2 19028.044} C_VEL
LIN {X 0,Y 405.527,Z 709.643,A -85,B 0,C 180,E1 19026.454,E2 19026.454} C_VEL
LIN {X 0,Y 402.174,Z 728.488,A -85,B 0,C 180,E1 19024.622,E2 19024.622} C_VEL
LIN {X 0,Y 398.89,Z 746.101,A -85,B 0,C 180,E1 19022.608,E2 19022.608} C_VEL
LIN {X 0,Y 395.843,Z 762.231,A -85,B 0,C 180,E1 19020.428,E2 19020.428} C_VEL
LIN {X 0,Y 392.861,Z 778.01,A -85,B 0,C 180,E1 19017.921,E2 19017.921} C_VEL
LIN {X 0,Y 390.213,Z 792.729,A -85,B 0,C 180,E1 19015.171,E2 19015.171} C_VEL
LIN {X 0,Y 388.1,Z 805.545,A -85,B 0,C 180,E1 19012.347,E2 19012.347} C_VEL
LIN {X 0,Y 386.508,Z 816.346,A -85,B 0,C 180,E1 19009.492,E2 19009.492} C_VEL
LIN {X 0,Y 385.327,Z 826.016,A -85,B 0,C 180,E1 19006.428,E2 19006.428} C_VEL
LIN {X 0,Y 384.594,Z 833.881,A -85,B 0,C 180,E1 19003.377,E2 19003.377} C_VEL
LIN {X 0,Y 384.224,Z 839.895,A -85,B 0,C 180,E1 19000.342,E2 19000.342} C_VEL
LIN {X 0,Y 384.081,Z 844.538,A -85,B 0,C 180,E1 18997.177,E2 18997.177} C_VEL
LIN {X 0,Y 384.054,Z 847.244,A -85,B 0,C 180,E1 18994.328,E2 18994.328} C_VEL
LIN {X 0,Y 384.074,Z 848.62,A -85,B 0,C 180,E1 18991.192,E2 18991.192} C_VEL
LIN {X 0,Y 384.076,Z 848.447,A -85,B 0,C 180,E1 18988.358,E2 18988.358} C_VEL
LIN {X 0,Y 384.08,Z 846.728,A -85,B 0,C 180,E1 18985.37,E2 18985.37} C_VEL
LIN {X 0,Y 384.108,Z 843.512,A -85,B 0,C 180,E1 18982.37,E2 18982.37} C_VEL
LIN {X 0,Y 384.29,Z 838.581,A -85,B 0,C 180,E1 18979.353,E2 18979.353} C_VEL
LIN {X 0,Y 384.681,Z 832.033,A -85,B 0,C 180,E1 18976.317,E2 18976.317} C_VEL
LIN {X 0,Y 385.382,Z 824.04,A -85,B 0,C 180,E1 18973.416,E2 18973.416} C_VEL
LIN {X 0,Y 386.536,Z 813.658,A -85,B 0,C 180,E1 18970.349,E2 18970.349} C_VEL
LIN {X 0,Y 388.009,Z 802.484,A -85,B 0,C 180,E1 18967.58,E2 18967.58} C_VEL
LIN {X 0,Y 389.959,Z 789.25,A -85,B 0,C 180,E1 18964.838,E2 18964.838} C_VEL
LIN {X 0,Y 392.368,Z 774.032,A -85,B 0,C 180,E1 18962.161,E2 18962.161} C_VEL
LIN {X 0,Y 395.155,Z 757.115,A -85,B 0,C 180,E1 18959.637,E2 18959.637} C_VEL
LIN {X 0,Y 398.12,Z 739.342,A -85,B 0,C 180,E1 18957.385,E2 18957.385} C_VEL
LIN {X 0,Y 401.185,Z 720.501,A -85,B 0,C 180,E1 18955.372,E2 18955.372} C_VEL
LIN {X 0,Y 404.416,Z 699.934,A -85,B 0,C 180,E1 18953.515,E2 18953.515} C_VEL
LIN {X 0,Y 407.603,Z 678.513,A -85,B 0,C 180,E1 18951.906,E2 18951.906} C_VEL
LIN {X 0,Y 410.674,Z 656.46,A -85,B 0,C 180,E1 18950.545,E2 18950.545} C_VEL
LIN {X 0,Y 413.519,Z 633.621,A -85,B 0,C 180,E1 18949.425,E2 18949.425} C_VEL
LIN {X 0,Y 416.124,Z 609.617,A -85,B 0,C 180,E1 18948.526,E2 18948.526} C_VEL
LIN {X 0,Y 418.138,Z 584.721,A -85,B 0,C 180,E1 18947.833,E2 18947.833} C_VEL
LIN {X 0,Y 423.581,Z 495.278,A -85,B 0,C 180,E1 18945.776,E2 18945.776} C_VEL
LIN {X 0,Y 430.041,Z 417.94,A -85,B 0,C 180,E1 18943.853,E2 18943.853} C_VEL
LIN {X 0,Y 437.727,Z 346.254,A -85,B 0,C 180,E1 18941.957,E2 18941.957} C_VEL
LIN {X 0,Y 437.692,Z 341.329,A -85,B 0,C 180,E1 18941.643,E2 18941.643} C_VEL
LIN {X 0,Y 435.872,Z 333.555,A -85,B 0,C 180,E1 18940.481,E2 18940.481} C_VEL
LIN {X 0,Y 434.695,Z 328.28,A -85,B 0,C 180,E1 18939.452,E2 18939.452} C_VEL
LIN {X 0,Y 433.863,Z 323.492,A -85,B 0,C 180,E1 18938.144,E2 18938.144} C_VEL
LIN {X 0,Y 433.727,Z 321.146,A -85,B 0,C 180,E1 18937.095,E2 18937.095} C_VEL
LIN {X 0,Y 434.341,Z 319.981,A -85,B 0,C 180,E1 18935.647,E2 18935.647} C_VEL
LIN {X 0,Y 435.565,Z 323.155,A -85,B 0,C 180,E1 18934.18,E2 18934.18} C_VEL
LIN {X 0,Y 437.336,Z 327.645,A -85,B 0,C 180,E1 18932.959,E2 18932.959} C_VEL
LIN {X 0,Y 438.802,Z 331.69,A -85,B 0,C 180,E1 18932.17,E2 18932.17} C_VEL
LIN {X 0,Y 430.762,Z 400.874,A -85,B 0,C 180,E1 18930.347,E2 18930.347} C_VEL
LIN {X 0,Y 424.538,Z 470.702,A -85,B 0,C 180,E1 18928.591,E2 18928.591} C_VEL
LIN {X 0,Y 419.172,Z 550.85,A -85,B 0,C 180,E1 18926.659,E2 18926.659} C_VEL
LIN {X 0,Y 417.344,Z 573.428,A -85,B 0,C 180,E1 18925.852,E2 18925.852} C_VEL
LIN {X 0,Y 415.081,Z 594.44,A -85,B 0,C 180,E1 18924.857,E2 18924.857} C_VEL
LIN {X 0,Y 412.485,Z 614.638,A -85,B 0,C 180,E1 18923.653,E2 18923.653} C_VEL
LIN {X 0,Y 409.447,Z 634.917,A -85,B 0,C 180,E1 18922.167,E2 18922.167} C_VEL
LIN {X 0,Y 406.376,Z 653.448,A -85,B 0,C 180,E1 18920.526,E2 18920.526} C_VEL
LIN {X 0,Y 403.02,Z 671.511,A -85,B 0,C 180,E1 18918.609,E2 18918.609} C_VEL
LIN {X 0,Y 399.817,Z 687.629,A -85,B 0,C 180,E1 18916.566,E2 18916.566} C_VEL
LIN {X 0,Y 396.678,Z 702.844,A -85,B 0,C 180,E1 18914.303,E2 18914.303} C_VEL
LIN {X 0,Y 393.798,Z 716.724,A -85,B 0,C 180,E1 18911.87,E2 18911.87} C_VEL
LIN {X 0,Y 391.19,Z 729.137,A -85,B 0,C 180,E1 18909.268,E2 18909.268} C_VEL
LIN {X 0,Y 388.863,Z 740.838,A -85,B 0,C 180,E1 18906.35,E2 18906.35} C_VEL
LIN {X 0,Y 387.098,Z 750.603,A -85,B 0,C 180,E1 18903.408,E2 18903.408} C_VEL
LIN {X 0,Y 385.783,Z 758.976,A -85,B 0,C 180,E1 18900.299,E2 18900.299} C_VEL
LIN {X 0,Y 384.914,Z 765.544,A -85,B 0,C 180,E1 18897.173,E2 18897.173} C_VEL
LIN {X 0,Y 384.421,Z 770.732,A -85,B 0,C 180,E1 18893.881,E2 18893.881} C_VEL
LIN {X 0,Y 384.192,Z 774.175,A -85,B 0,C 180,E1 18890.717,E2 18890.717} C_VEL
LIN {X 0,Y 384.096,Z 775.996,A -85,B 0,C 180,E1 18887.525,E2 18887.525} C_VEL
LIN {X 0,Y 384.085,Z 776.352,A -85,B 0,C 180,E1 18884.294,E2 18884.294} C_VEL
LIN {X 0,Y 384.107,Z 775.261,A -85,B 0,C 180,E1 18881.171,E2 18881.171} C_VEL
LIN {X 0,Y 384.203,Z 772.554,A -85,B 0,C 180,E1 18877.994,E2 18877.994} C_VEL
LIN {X 0,Y 384.487,Z 768.262,A -85,B 0,C 180,E1 18874.758,E2 18874.758} C_VEL
LIN {X 0,Y 385.059,Z 762.533,A -85,B 0,C 180,E1 18871.632,E2 18871.632} C_VEL
LIN {X 0,Y 385.966,Z 755.333,A -85,B 0,C 180,E1 18868.624,E2 18868.624} C_VEL
LIN {X 0,Y 387.455,Z 745.785,A -85,B 0,C 180,E1 18865.408,E2 18865.408} C_VEL
LIN {X 0,Y 389.353,Z 735.331,A -85,B 0,C 180,E1 18862.514,E2 18862.514} C_VEL
LIN {X 0,Y 391.672,Z 723.313,A -85,B 0,C 180,E1 18859.756,E2 18859.756} C_VEL
LIN {X 0,Y 394.437,Z 709.62,A -85,B 0,C 180,E1 18857.105,E2 18857.105} C_VEL
LIN {X 0,Y 397.555,Z 694.507,A -85,B 0,C 180,E1 18854.627,E2 18854.627} C_VEL
LIN {X 0,Y 400.687,Z 679.053,A -85,B 0,C 180,E1 18852.481,E2 18852.481} C_VEL
LIN {X 0,Y 403.975,Z 661.958,A -85,B 0,C 180,E1 18850.476,E2 18850.476} C_VEL
LIN {X 0,Y 407.433,Z 642.845,A -85,B 0,C 180,E1 18848.585,E2 18848.585} C_VEL
LIN {X 0,Y 410.634,Z 623.703,A -85,B 0,C 180,E1 18847.003,E2 18847.003} C_VEL
LIN {X 0,Y 413.556,Z 603.479,A -85,B 0,C 180,E1 18845.64,E2 18845.64} C_VEL
LIN {X 0,Y 416.126,Z 582.625,A -85,B 0,C 180,E1 18844.503,E2 18844.503} C_VEL
LIN {X 0,Y 418.344,Z 560.958,A -85,B 0,C 180,E1 18843.581,E2 18843.581} C_VEL
LIN {X 0,Y 419.976,Z 539.838,A -85,B 0,C 180,E1 18842.922,E2 18842.922} C_VEL
LIN {X 0,Y 421.615,Z 504.552,A -85,B 0,C 180,E1 18842.181,E2 18842.181} C_VEL
LIN {X 0,Y 429.56,Z 328.497,A -85,B 0,C 180,E1 18838.672,E2 18838.672} C_VEL
LIN {X 0,Y 416.785,Z 309.164,A -85,B 0,C 180,E1 18836.406,E2 18836.406} C_VEL
LIN {X 0,Y 403.555,Z 290.347,A -85,B 0,C 180,E1 18833.859,E2 18833.859} C_VEL
LIN {X 0,Y 395.889,Z 279.888,A -85,B 0,C 180,E1 18832.263,E2 18832.263} C_VEL
LIN {X 0,Y 392.761,Z 275.552,A -85,B 0,C 180,E1 18831.585,E2 18831.585} C_VEL
LIN {X 0,Y 389.998,Z 271.822,A -85,B 0,C 180,E1 18830.976,E2 18830.976} C_VEL
LIN {X 0,Y 389.117,Z 270.366,A -85,B 0,C 180,E1 18830.77,E2 18830.77} C_VEL
LIN {X 0,Y 386.582,Z 267.682,A -85,B 0,C 180,E1 18830.22,E2 18830.22} C_VEL
LIN {X 0,Y 385.592,Z 264.705,A -85,B 0,C 180,E1 18829.899,E2 18829.899} C_VEL
LIN {X 0,Y 385.59,Z 264.7,A -85,B 0,C 180,E1 18825.853,E2 18825.853} C_VEL
LIN {X 0,Y 385.625,Z 264.701,A -85,B 0,C 180,E1 18825.168,E2 18825.168} C_VEL
LIN {X 0,Y 384.664,Z 264.828,A -85,B 0,C 180,E1 18824.023,E2 18824.023} C_VEL
LIN {X 0,Y 379.866,Z 265.425,A -85,B 0,C 180,E1 18821.783,E2 18821.783} C_VEL
LIN {X 0,Y 377.792,Z 265.678,A -85,B 0,C 180,E1 18820.375,E2 18820.375} C_VEL
LIN {X 0,Y 377.647,Z 265.694,A -85,B 0,C 180,E1 18819.951,E2 18819.951} C_VEL
LIN {X 0,Y 377.645,Z 265.686,A -85,B 0,C 180,E1 18815.928,E2 18815.928} C_VEL
LIN {X 0,Y 377.643,Z 265.684,A -85,B 0,C 180,E1 18811.822,E2 18811.822} C_VEL
LIN {X 0,Y 377.642,Z 265.689,A -85,B 0,C 180,E1 18807.725,E2 18807.725} C_VEL
LIN {X 0,Y 377.641,Z 265.689,A -85,B 0,C 180,E1 18803.617,E2 18803.617} C_VEL
LIN {X 0,Y 377.64,Z 265.689,A -85,B 0,C 180,E1 18799.63,E2 18799.63} C_VEL
LIN {X 0,Y 377.638,Z 265.69,A -85,B 0,C 180,E1 18795.59,E2 18795.59} C_VEL
LIN {X 0,Y 377.638,Z 265.691,A -85,B 0,C 180,E1 18791.477,E2 18791.477} C_VEL
LIN {X 0,Y 377.636,Z 265.692,A -85,B 0,C 180,E1 18787.426,E2 18787.426} C_VEL
LIN {X 0,Y 377.636,Z 265.694,A -85,B 0,C 180,E1 18783.421,E2 18783.421} C_VEL
LIN {X 0,Y 377.633,Z 265.696,A -85,B 0,C 180,E1 18779.367,E2 18779.367} C_VEL
LIN {X 0,Y 377.63,Z 265.697,A -85,B 0,C 180,E1 18775.304,E2 18775.304} C_VEL
LIN {X 0,Y 377.63,Z 265.698,A -85,B 0,C 180,E1 18771.33,E2 18771.33} C_VEL
LIN {X 0,Y 377.629,Z 265.697,A -85,B 0,C 180,E1 18767.329,E2 18767.329} C_VEL
LIN {X 0,Y 377.627,Z 265.692,A -85,B 0,C 180,E1 18763.273,E2 18763.273} C_VEL
LIN {X 0,Y 377.627,Z 265.687,A -85,B 0,C 180,E1 18759.254,E2 18759.254} C_VEL
LIN {X 0,Y 377.626,Z 265.687,A -85,B 0,C 180,E1 18755.251,E2 18755.251} C_VEL
LIN {X 0,Y 377.625,Z 265.691,A -85,B 0,C 180,E1 18751.22,E2 18751.22} C_VEL
LIN {X 0,Y 377.627,Z 265.694,A -85,B 0,C 180,E1 18747.259,E2 18747.259} C_VEL
LIN {X 0,Y 377.628,Z 265.695,A -85,B 0,C 180,E1 18743.233,E2 18743.233} C_VEL
LIN {X 0,Y 377.633,Z 265.695,A -85,B 0,C 180,E1 18739.325,E2 18739.325} C_VEL
LIN {X 0,Y 377.635,Z 265.694,A -85,B 0,C 180,E1 18735.351,E2 18735.351} C_VEL
LIN {X 0,Y 377.645,Z 265.69,A -85,B 0,C 180,E1 18731.451,E2 18731.451} C_VEL
LIN {X 0,Y 377.65,Z 265.688,A -85,B 0,C 180,E1 18727.452,E2 18727.452} C_VEL
LIN {X 0,Y 377.641,Z 265.691,A -85,B 0,C 180,E1 18723.337,E2 18723.337} C_VEL
LIN {X 0,Y 377.656,Z 265.694,A -85,B 0,C 180,E1 18719.391,E2 18719.391} C_VEL
LIN {X 0,Y 377.649,Z 265.691,A -85,B 0,C 180,E1 18715.29,E2 18715.29} C_VEL
LIN {X 0,Y 377.659,Z 265.688,A -85,B 0,C 180,E1 18711.319,E2 18711.319} C_VEL
LIN {X 0,Y 377.655,Z 265.692,A -85,B 0,C 180,E1 18707.149,E2 18707.149} C_VEL
LIN {X 0,Y 377.661,Z 265.687,A -85,B 0,C 180,E1 18703.225,E2 18703.225} C_VEL
LIN {X 0,Y 377.66,Z 265.686,A -85,B 0,C 180,E1 18699.057,E2 18699.057} C_VEL
LIN {X 0,Y 377.663,Z 265.688,A -85,B 0,C 180,E1 18695.104,E2 18695.104} C_VEL
LIN {X 0,Y 377.671,Z 265.688,A -85,B 0,C 180,E1 18690.993,E2 18690.993} C_VEL
LIN {X 0,Y 378.762,Z 268.913,A -85,B 0,C 180,E1 18690.244,E2 18690.244} C_VEL
LIN {X 0,Y 380.194,Z 271,A -85,B 0,C 180,E1 18689.672,E2 18689.672} C_VEL
LIN {X 0,Y 387.294,Z 284.95,A -85,B 0,C 180,E1 18686.462,E2 18686.462} C_VEL
LIN {X 0,Y 390.438,Z 291.161,A -85,B 0,C 180,E1 18685.174,E2 18685.174} C_VEL
LIN {X 0,Y 401.028,Z 307.018,A -85,B 0,C 180,E1 18682.843,E2 18682.843} C_VEL
LIN {X 0,Y 414.147,Z 327.711,A -85,B 0,C 180,E1 18680.178,E2 18680.178} C_VEL
LIN {X 0,Y 425.255,Z 346.631,A -85,B 0,C 180,E1 18678.069,E2 18678.069} C_VEL
LIN {X 0,Y 416.577,Z 524.513,A -85,B 0,C 180,E1 18674.435,E2 18674.435} C_VEL
LIN {X 0,Y 413.022,Z 602.36,A -85,B 0,C 180,E1 18672.84,E2 18672.84} C_VEL
LIN {X 0,Y 410.915,Z 625.303,A -85,B 0,C 180,E1 18672.151,E2 18672.151} C_VEL
LIN {X 0,Y 408.349,Z 647.081,A -85,B 0,C 180,E1 18671.246,E2 18671.246} C_VEL
LIN {X 0,Y 405.232,Z 669.693,A -85,B 0,C 180,E1 18670.021,E2 18670.021} C_VEL
LIN {X 0,Y 402.127,Z 689.288,A -85,B 0,C 180,E1 18668.704,E2 18668.704} C_VEL
LIN {X 0,Y 398.515,Z 709.682,A -85,B 0,C 180,E1 18667.022,E2 18667.022} C_VEL
LIN {X 0,Y 394.995,Z 728.522,A -85,B 0,C 180,E1 18665.152,E2 18665.152} C_VEL
LIN {X 0,Y 391.348,Z 747.095,A -85,B 0,C 180,E1 18662.968,E2 18662.968} C_VEL
LIN {X 0,Y 388.095,Z 763.662,A -85,B 0,C 180,E1 18660.669,E2 18660.669} C_VEL
LIN {X 0,Y 385.114,Z 778.721,A -85,B 0,C 180,E1 18658.196,E2 18658.196} C_VEL
LIN {X 0,Y 382.369,Z 793.229,A -85,B 0,C 180,E1 18655.392,E2 18655.392} C_VEL
LIN {X 0,Y 380.224,Z 805.598,A -85,B 0,C 180,E1 18652.575,E2 18652.575} C_VEL
LIN {X 0,Y 378.542,Z 816.554,A -85,B 0,C 180,E1 18649.598,E2 18649.598} C_VEL
LIN {X 0,Y 377.331,Z 826.055,A -85,B 0,C 180,E1 18646.469,E2 18646.469} C_VEL
LIN {X 0,Y 376.592,Z 833.754,A -85,B 0,C 180,E1 18643.353,E2 18643.353} C_VEL
LIN {X 0,Y 376.239,Z 839.409,A -85,B 0,C 180,E1 18640.409,E2 18640.409} C_VEL
LIN {X 0,Y 376.101,Z 843.965,A -85,B 0,C 180,E1 18637.176,E2 18637.176} C_VEL
LIN {X 0,Y 376.081,Z 846.622,A -85,B 0,C 180,E1 18634.268,E2 18634.268} C_VEL
LIN {X 0,Y 376.109,Z 847.87,A -85,B 0,C 180,E1 18631.217,E2 18631.217} C_VEL
LIN {X 0,Y 376.112,Z 847.716,A -85,B 0,C 180,E1 18628.475,E2 18628.475} C_VEL
LIN {X 0,Y 376.111,Z 846.054,A -85,B 0,C 180,E1 18625.424,E2 18625.424} C_VEL
LIN {X 0,Y 376.132,Z 843.051,A -85,B 0,C 180,E1 18622.514,E2 18622.514} C_VEL
LIN {X 0,Y 376.298,Z 838.269,A -85,B 0,C 180,E1 18619.434,E2 18619.434} C_VEL
LIN {X 0,Y 376.679,Z 831.846,A -85,B 0,C 180,E1 18616.334,E2 18616.334} C_VEL
LIN {X 0,Y 377.388,Z 823.917,A -85,B 0,C 180,E1 18613.372,E2 18613.372} C_VEL
LIN {X 0,Y 378.569,Z 813.709,A -85,B 0,C 180,E1 18610.24,E2 18610.24} C_VEL
LIN {X 0,Y 380.186,Z 801.966,A -85,B 0,C 180,E1 18607.256,E2 18607.256} C_VEL
LIN {X 0,Y 382.253,Z 788.611,A -85,B 0,C 180,E1 18604.43,E2 18604.43} C_VEL
LIN {X 0,Y 384.792,Z 773.394,A -85,B 0,C 180,E1 18601.699,E2 18601.699} C_VEL
LIN {X 0,Y 387.541,Z 757.585,A -85,B 0,C 180,E1 18599.279,E2 18599.279} C_VEL
LIN {X 0,Y 390.547,Z 740.414,A -85,B 0,C 180,E1 18597.04,E2 18597.04} C_VEL
LIN {X 0,Y 393.889,Z 721.078,A -85,B 0,C 180,E1 18594.902,E2 18594.902} C_VEL
LIN {X 0,Y 397.412,Z 699.962,A -85,B 0,C 180,E1 18592.945,E2 18592.945} C_VEL
LIN {X 0,Y 400.738,Z 679.016,A -85,B 0,C 180,E1 18591.325,E2 18591.325} C_VEL
LIN {X 0,Y 404.084,Z 656.477,A -85,B 0,C 180,E1 18589.897,E2 18589.897} C_VEL
LIN {X 0,Y 407.155,Z 633.484,A -85,B 0,C 180,E1 18588.738,E2 18588.738} C_VEL
LIN {X 0,Y 410.051,Z 608.923,A -85,B 0,C 180,E1 18587.789,E2 18587.789} C_VEL
LIN {X 0,Y 412.309,Z 583.43,A -85,B 0,C 180,E1 18587.054,E2 18587.054} C_VEL
LIN {X 0,Y 418.213,Z 497.754,A -85,B 0,C 180,E1 18585.001,E2 18585.001} C_VEL
LIN {X 0,Y 425.114,Z 423.935,A -85,B 0,C 180,E1 18583.101,E2 18583.101} C_VEL
LIN {X 0,Y 433.794,Z 351.926,A -85,B 0,C 180,E1 18581.162,E2 18581.162} C_VEL
LIN {X 0,Y 434.263,Z 347.428,A -85,B 0,C 180,E1 18580.994,E2 18580.994} C_VEL
LIN {X 0,Y 434.196,Z 345.7,A -85,B 0,C 180,E1 18580.844,E2 18580.844} C_VEL
LIN {X 0,Y 433.004,Z 338.896,A -85,B 0,C 180,E1 18579.765,E2 18579.765} C_VEL
LIN {X 0,Y 432.137,Z 333.108,A -85,B 0,C 180,E1 18578.493,E2 18578.493} C_VEL
LIN {X 0,Y 431.93,Z 329.709,A -85,B 0,C 180,E1 18577.338,E2 18577.338} C_VEL
LIN {X 0,Y 432.091,Z 328.502,A -85,B 0,C 180,E1 18576.585,E2 18576.585} C_VEL
LIN {X 0,Y 432.581,Z 327.932,A -85,B 0,C 180,E1 18575.707,E2 18575.707} C_VEL
LIN {X 0,Y 433.479,Z 330.775,A -85,B 0,C 180,E1 18574.411,E2 18574.411} C_VEL
LIN {X 0,Y 434.96,Z 335.108,A -85,B 0,C 180,E1 18573.24,E2 18573.24} C_VEL
LIN {X 0,Y 435.223,Z 336.447,A -85,B 0,C 180,E1 18573.029,E2 18573.029} C_VEL
LIN {X 0,Y 426.02,Z 407.277,A -85,B 0,C 180,E1 18571.108,E2 18571.108} C_VEL
LIN {X 0,Y 419.228,Z 475.229,A -85,B 0,C 180,E1 18569.34,E2 18569.34} C_VEL
LIN {X 0,Y 413.42,Z 552.438,A -85,B 0,C 180,E1 18567.4,E2 18567.4} C_VEL
LIN {X 0,Y 411.413,Z 575.057,A -85,B 0,C 180,E1 18566.564,E2 18566.564} C_VEL
LIN {X 0,Y 408.948,Z 596.268,A -85,B 0,C 180,E1 18565.531,E2 18565.531} C_VEL
LIN {X 0,Y 406.134,Z 616.714,A -85,B 0,C 180,E1 18564.278,E2 18564.278} C_VEL
LIN {X 0,Y 402.944,Z 636.7,A -85,B 0,C 180,E1 18562.775,E2 18562.775} C_VEL
LIN {X 0,Y 399.708,Z 655.001,A -85,B 0,C 180,E1 18561.115,E2 18561.115} C_VEL
LIN {X 0,Y 396.283,Z 672.479,A -85,B 0,C 180,E1 18559.226,E2 18559.226} C_VEL
LIN {X 0,Y 392.825,Z 688.985,A -85,B 0,C 180,E1 18557.098,E2 18557.098} C_VEL
LIN {X 0,Y 389.419,Z 704.522,A -85,B 0,C 180,E1 18554.727,E2 18554.727} C_VEL
LIN {X 0,Y 386.395,Z 718.283,A -85,B 0,C 180,E1 18552.252,E2 18552.252} C_VEL
LIN {X 0,Y 383.523,Z 731.261,A -85,B 0,C 180,E1 18549.455,E2 18549.455} C_VEL
LIN {X 0,Y 381.198,Z 742.185,A -85,B 0,C 180,E1 18546.629,E2 18546.629} C_VEL
LIN {X 0,Y 379.247,Z 752.273,A -85,B 0,C 180,E1 18543.478,E2 18543.478} C_VEL
LIN {X 0,Y 377.938,Z 760.158,A -85,B 0,C 180,E1 18540.457,E2 18540.457} C_VEL
LIN {X 0,Y 377.011,Z 766.623,A -85,B 0,C 180,E1 18537.266,E2 18537.266} C_VEL
LIN {X 0,Y 376.482,Z 771.724,A -85,B 0,C 180,E1 18533.904,E2 18533.904} C_VEL
LIN {X 0,Y 376.234,Z 775.071,A -85,B 0,C 180,E1 18530.673,E2 18530.673} C_VEL
LIN {X 0,Y 376.135,Z 776.766,A -85,B 0,C 180,E1 18527.568,E2 18527.568} C_VEL
LIN {X 0,Y 376.12,Z 777.083,A -85,B 0,C 180,E1 18524.224,E2 18524.224} C_VEL
LIN {X 0,Y 376.145,Z 775.978,A -85,B 0,C 180,E1 18521.08,E2 18521.08} C_VEL
LIN {X 0,Y 376.243,Z 773.395,A -85,B 0,C 180,E1 18517.997,E2 18517.997} C_VEL
LIN {X 0,Y 376.548,Z 769.149,A -85,B 0,C 180,E1 18514.693,E2 18514.693} C_VEL
LIN {X 0,Y 377.151,Z 763.432,A -85,B 0,C 180,E1 18511.501,E2 18511.501} C_VEL
LIN {X 0,Y 378.138,Z 756.113,A -85,B 0,C 180,E1 18508.368,E2 18508.368} C_VEL
LIN {X 0,Y 379.686,Z 746.768,A -85,B 0,C 180,E1 18505.152,E2 18505.152} C_VEL
LIN {X 0,Y 381.684,Z 736.334,A -85,B 0,C 180,E1 18502.198,E2 18502.198} C_VEL
LIN {X 0,Y 384.152,Z 724.164,A -85,B 0,C 180,E1 18499.351,E2 18499.351} C_VEL
LIN {X 0,Y 387.044,Z 710.514,A -85,B 0,C 180,E1 18496.662,E2 18496.662} C_VEL
LIN {X 0,Y 390.262,Z 695.548,A -85,B 0,C 180,E1 18494.167,E2 18494.167} C_VEL
LIN {X 0,Y 393.646,Z 679.534,A -85,B 0,C 180,E1 18491.912,E2 18491.912} C_VEL
LIN {X 0,Y 397.141,Z 662.074,A -85,B 0,C 180,E1 18489.841,E2 18489.841} C_VEL
LIN {X 0,Y 400.811,Z 642.577,A -85,B 0,C 180,E1 18487.901,E2 18487.901} C_VEL
LIN {X 0,Y 404.046,Z 623.912,A -85,B 0,C 180,E1 18486.348,E2 18486.348} C_VEL
LIN {X 0,Y 407.026,Z 604.1,A -85,B 0,C 180,E1 18484.996,E2 18484.996} C_VEL
LIN {X 0,Y 409.686,Z 583.332,A -85,B 0,C 180,E1 18483.851,E2 18483.851} C_VEL
LIN {X 0,Y 411.993,Z 561.575,A -85,B 0,C 180,E1 18482.915,E2 18482.915} C_VEL
LIN {X 0,Y 413.693,Z 540.328,A -85,B 0,C 180,E1 18482.244,E2 18482.244} C_VEL
LIN {X 0,Y 415.508,Z 503.122,A -85,B 0,C 180,E1 18481.453,E2 18481.453} C_VEL
LIN {X 0,Y 423.573,Z 331.936,A -85,B 0,C 180,E1 18477.994,E2 18477.994} C_VEL
LIN {X 0,Y 409.703,Z 311.02,A -85,B 0,C 180,E1 18475.438,E2 18475.438} C_VEL
LIN {X 0,Y 396.341,Z 292.075,A -85,B 0,C 180,E1 18472.745,E2 18472.745} C_VEL
LIN {X 0,Y 388.729,Z 281.769,A -85,B 0,C 180,E1 18471.107,E2 18471.107} C_VEL
LIN {X 0,Y 384.953,Z 276.624,A -85,B 0,C 180,E1 18470.25,E2 18470.25} C_VEL
LIN {X 0,Y 382.168,Z 272.963,A -85,B 0,C 180,E1 18469.607,E2 18469.607} C_VEL
LIN {X 0,Y 381.246,Z 271.402,A -85,B 0,C 180,E1 18469.377,E2 18469.377} C_VEL
LIN {X 0,Y 378.632,Z 268.602,A -85,B 0,C 180,E1 18468.775,E2 18468.775} C_VEL
LIN {X 0,Y 377.659,Z 265.687,A -85,B 0,C 180,E1 18468.447,E2 18468.447} C_VEL
LIN {X 0,Y 377.657,Z 265.688,A -85,B 0,C 180,E1 18464.412,E2 18464.412} C_VEL
LIN {X 0,Y 377.658,Z 265.69,A -85,B 0,C 180,E1 18460.373,E2 18460.373} C_VEL
LIN {X 0,Y 377.647,Z 265.694,A -85,B 0,C 180,E1 18459.951,E2 18459.951} C_VEL
LIN {X 0,Y 376.674,Z 265.814,A -85,B 0,C 180,E1 18458.783,E2 18458.783} C_VEL
LIN {X 0,Y 370.108,Z 266.623,A -85,B 0,C 180,E1 18455.312,E2 18455.312} C_VEL
LIN {X 0,Y 369.733,Z 266.672,A -85,B 0,C 180,E1 18454.621,E2 18454.621} C_VEL
LIN {X 0,Y 369.73,Z 266.676,A -85,B 0,C 180,E1 18450.466,E2 18450.466} C_VEL
LIN {X 0,Y 369.727,Z 266.669,A -85,B 0,C 180,E1 18446.436,E2 18446.436} C_VEL
LIN {X 0,Y 369.732,Z 266.667,A -85,B 0,C 180,E1 18442.387,E2 18442.387} C_VEL
LIN {X 0,Y 369.724,Z 266.669,A -85,B 0,C 180,E1 18438.299,E2 18438.299} C_VEL
LIN {X 0,Y 369.727,Z 266.669,A -85,B 0,C 180,E1 18434.297,E2 18434.297} C_VEL
LIN {X 0,Y 369.725,Z 266.67,A -85,B 0,C 180,E1 18430.228,E2 18430.228} C_VEL
LIN {X 0,Y 369.729,Z 266.67,A -85,B 0,C 180,E1 18426.24,E2 18426.24} C_VEL
LIN {X 0,Y 369.723,Z 266.671,A -85,B 0,C 180,E1 18422.107,E2 18422.107} C_VEL
LIN {X 0,Y 369.724,Z 266.673,A -85,B 0,C 180,E1 18418.114,E2 18418.114} C_VEL
LIN {X 0,Y 369.715,Z 266.677,A -85,B 0,C 180,E1 18413.955,E2 18413.955} C_VEL
LIN {X 0,Y 369.72,Z 266.682,A -85,B 0,C 180,E1 18409.932,E2 18409.932} C_VEL
LIN {X 0,Y 369.722,Z 266.686,A -85,B 0,C 180,E1 18405.974,E2 18405.974} C_VEL
LIN {X 0,Y 369.723,Z 266.687,A -85,B 0,C 180,E1 18401.907,E2 18401.907} C_VEL
LIN {X 0,Y 369.721,Z 266.682,A -85,B 0,C 180,E1 18397.849,E2 18397.849} C_VEL
LIN {X 0,Y 369.72,Z 266.675,A -85,B 0,C 180,E1 18393.852,E2 18393.852} C_VEL
LIN {X 0,Y 369.721,Z 266.672,A -85,B 0,C 180,E1 18389.766,E2 18389.766} C_VEL
LIN {X 0,Y 369.719,Z 266.67,A -85,B 0,C 180,E1 18385.774,E2 18385.774} C_VEL
LIN {X 0,Y 369.726,Z 266.673,A -85,B 0,C 180,E1 18381.743,E2 18381.743} C_VEL
LIN {X 0,Y 369.714,Z 266.675,A -85,B 0,C 180,E1 18377.629,E2 18377.629} C_VEL
LIN {X 0,Y 369.718,Z 266.676,A -85,B 0,C 180,E1 18373.606,E2 18373.606} C_VEL
LIN {X 0,Y 369.708,Z 266.682,A -85,B 0,C 180,E1 18369.493,E2 18369.493} C_VEL
LIN {X 0,Y 369.708,Z 266.686,A -85,B 0,C 180,E1 18365.429,E2 18365.429} C_VEL
LIN {X 0,Y 369.698,Z 266.679,A -85,B 0,C 180,E1 18361.238,E2 18361.238} C_VEL
LIN {X 0,Y 369.701,Z 266.679,A -85,B 0,C 180,E1 18357.208,E2 18357.208} C_VEL
LIN {X 0,Y 369.706,Z 266.685,A -85,B 0,C 180,E1 18353.164,E2 18353.164} C_VEL
LIN {X 0,Y 369.704,Z 266.678,A -85,B 0,C 180,E1 18349.085,E2 18349.085} C_VEL
LIN {X 0,Y 369.717,Z 266.682,A -85,B 0,C 180,E1 18345.111,E2 18345.111} C_VEL
LIN {X 0,Y 369.716,Z 266.675,A -85,B 0,C 180,E1 18341.061,E2 18341.061} C_VEL
LIN {X 0,Y 369.713,Z 266.675,A -85,B 0,C 180,E1 18336.911,E2 18336.911} C_VEL
LIN {X 0,Y 369.711,Z 266.677,A -85,B 0,C 180,E1 18332.802,E2 18332.802} C_VEL
LIN {X 0,Y 369.705,Z 266.792,A -85,B 0,C 180,E1 18332.408,E2 18332.408} C_VEL
LIN {X 0,Y 370.902,Z 270.015,A -85,B 0,C 180,E1 18331.675,E2 18331.675} C_VEL
LIN {X 0,Y 372.292,Z 272.031,A -85,B 0,C 180,E1 18331.089,E2 18331.089} C_VEL
LIN {X 0,Y 374.11,Z 275.672,A -85,B 0,C 180,E1 18330.19,E2 18330.19} C_VEL
LIN {X 0,Y 379.868,Z 286.917,A -85,B 0,C 180,E1 18327.522,E2 18327.522} C_VEL
LIN {X 0,Y 381.874,Z 290.498,A -85,B 0,C 180,E1 18326.755,E2 18326.755} C_VEL
LIN {X 0,Y 395.689,Z 310.989,A -85,B 0,C 180,E1 18323.593,E2 18323.593} C_VEL
LIN {X 0,Y 410.114,Z 334.087,A -85,B 0,C 180,E1 18320.571,E2 18320.571} C_VEL
LIN {X 0,Y 419.469,Z 350.299,A -85,B 0,C 180,E1 18318.755,E2 18318.755} C_VEL
LIN {X 0,Y 409.813,Z 538.426,A -85,B 0,C 180,E1 18314.872,E2 18314.872} C_VEL
LIN {X 0,Y 406.667,Z 602.36,A -85,B 0,C 180,E1 18313.521,E2 18313.521} C_VEL
LIN {X 0,Y 404.482,Z 625.171,A -85,B 0,C 180,E1 18312.824,E2 18312.824} C_VEL
LIN {X 0,Y 401.752,Z 647.272,A -85,B 0,C 180,E1 18311.889,E2 18311.889} C_VEL
LIN {X 0,Y 398.535,Z 669.57,A -85,B 0,C 180,E1 18310.659,E2 18310.659} C_VEL
LIN {X 0,Y 395.153,Z 689.965,A -85,B 0,C 180,E1 18309.259,E2 18309.259} C_VEL
LIN {X 0,Y 391.538,Z 709.651,A -85,B 0,C 180,E1 18307.611,E2 18307.611} C_VEL
LIN {X 0,Y 388.022,Z 727.692,A -85,B 0,C 180,E1 18305.796,E2 18305.796} C_VEL
LIN {X 0,Y 384.284,Z 745.899,A -85,B 0,C 180,E1 18303.632,E2 18303.632} C_VEL
LIN {X 0,Y 380.772,Z 762.927,A -85,B 0,C 180,E1 18301.237,E2 18301.237} C_VEL
LIN {X 0,Y 377.54,Z 778.446,A -85,B 0,C 180,E1 18298.641,E2 18298.641} C_VEL
LIN {X 0,Y 374.81,Z 792.194,A -85,B 0,C 180,E1 18295.942,E2 18295.942} C_VEL
LIN {X 0,Y 372.527,Z 804.676,A -85,B 0,C 180,E1 18293.068,E2 18293.068} C_VEL
LIN {X 0,Y 370.738,Z 815.672,A -85,B 0,C 180,E1 18290.028,E2 18290.028} C_VEL
LIN {X 0,Y 369.442,Z 825.223,A -85,B 0,C 180,E1 18286.831,E2 18286.831} C_VEL
LIN {X 0,Y 368.643,Z 832.962,A -85,B 0,C 180,E1 18283.647,E2 18283.647} C_VEL
LIN {X 0,Y 368.267,Z 838.66,A -85,B 0,C 180,E1 18280.625,E2 18280.625} C_VEL
LIN {X 0,Y 368.116,Z 843.218,A -85,B 0,C 180,E1 18277.333,E2 18277.333} C_VEL
LIN {X 0,Y 368.109,Z 845.881,A -85,B 0,C 180,E1 18274.36,E2 18274.36} C_VEL
LIN {X 0,Y 368.142,Z 847.123,A -85,B 0,C 180,E1 18271.243,E2 18271.243} C_VEL
LIN {X 0,Y 368.147,Z 846.957,A -85,B 0,C 180,E1 18268.442,E2 18268.442} C_VEL
LIN {X 0,Y 368.143,Z 845.267,A -85,B 0,C 180,E1 18265.325,E2 18265.325} C_VEL
LIN {X 0,Y 368.158,Z 842.218,A -85,B 0,C 180,E1 18262.351,E2 18262.351} C_VEL
LIN {X 0,Y 368.327,Z 837.377,A -85,B 0,C 180,E1 18259.203,E2 18259.203} C_VEL
LIN {X 0,Y 368.721,Z 831.097,A -85,B 0,C 180,E1 18256.119,E2 18256.119} C_VEL
LIN {X 0,Y 369.502,Z 822.916,A -85,B 0,C 180,E1 18253.006,E2 18253.006} C_VEL
LIN {X 0,Y 370.761,Z 812.587,A -85,B 0,C 180,E1 18249.799,E2 18249.799} C_VEL
LIN {X 0,Y 372.376,Z 801.462,A -85,B 0,C 180,E1 18246.918,E2 18246.918} C_VEL
LIN {X 0,Y 374.545,Z 788.161,A -85,B 0,C 180,E1 18244.035,E2 18244.035} C_VEL
LIN {X 0,Y 377.222,Z 772.93,A -85,B 0,C 180,E1 18241.243,E2 18241.243} C_VEL
LIN {X 0,Y 380.159,Z 756.953,A -85,B 0,C 180,E1 18238.737,E2 18238.737} C_VEL
LIN {X 0,Y 383.615,Z 738.306,A -85,B 0,C 180,E1 18236.277,E2 18236.277} C_VEL
LIN {X 0,Y 387.165,Z 718.78,A -85,B 0,C 180,E1 18234.109,E2 18234.109} C_VEL
LIN {X 0,Y 390.767,Z 698.384,A -85,B 0,C 180,E1 18232.206,E2 18232.206} C_VEL
LIN {X 0,Y 394.131,Z 678.477,A -85,B 0,C 180,E1 18230.637,E2 18230.637} C_VEL
LIN {X 0,Y 397.7,Z 655.882,A -85,B 0,C 180,E1 18229.179,E2 18229.179} C_VEL
LIN {X 0,Y 401.003,Z 632.885,A -85,B 0,C 180,E1 18227.992,E2 18227.992} C_VEL
LIN {X 0,Y 404.235,Z 607.63,A -85,B 0,C 180,E1 18226.991,E2 18226.991} C_VEL
LIN {X 0,Y 406.717,Z 581.919,A -85,B 0,C 180,E1 18226.226,E2 18226.226} C_VEL
LIN {X 0,Y 413.205,Z 499.13,A -85,B 0,C 180,E1 18224.158,E2 18224.158} C_VEL
LIN {X 0,Y 420.795,Z 427.04,A -85,B 0,C 180,E1 18222.235,E2 18222.235} C_VEL
LIN {X 0,Y 430.625,Z 354.566,A -85,B 0,C 180,E1 18220.228,E2 18220.228} C_VEL
LIN {X 0,Y 431.18,Z 350.645,A -85,B 0,C 180,E1 18220.097,E2 18220.097} C_VEL
LIN {X 0,Y 430.439,Z 343.876,A -85,B 0,C 180,E1 18218.956,E2 18218.956} C_VEL
LIN {X 0,Y 430.132,Z 338.747,A -85,B 0,C 180,E1 18217.627,E2 18217.627} C_VEL
LIN {X 0,Y 430.341,Z 336.479,A -85,B 0,C 180,E1 18216.665,E2 18216.665} C_VEL
LIN {X 0,Y 430.816,Z 335.829,A -85,B 0,C 180,E1 18215.794,E2 18215.794} C_VEL
LIN {X 0,Y 431.44,Z 338.212,A -85,B 0,C 180,E1 18214.706,E2 18214.706} C_VEL
LIN {X 0,Y 432.157,Z 341.041,A -85,B 0,C 180,E1 18213.925,E2 18213.925} C_VEL
LIN {X 0,Y 422.5,Z 406.94,A -85,B 0,C 180,E1 18212.094,E2 18212.094} C_VEL
LIN {X 0,Y 414.937,Z 472.207,A -85,B 0,C 180,E1 18210.326,E2 18210.326} C_VEL
LIN {X 0,Y 407.911,Z 553.758,A -85,B 0,C 180,E1 18208.191,E2 18208.191} C_VEL
LIN {X 0,Y 405.698,Z 576.454,A -85,B 0,C 180,E1 18207.325,E2 18207.325} C_VEL
LIN {X 0,Y 403.074,Z 597.348,A -85,B 0,C 180,E1 18206.283,E2 18206.283} C_VEL
LIN {X 0,Y 400.187,Z 617.052,A -85,B 0,C 180,E1 18205.057,E2 18205.057} C_VEL
LIN {X 0,Y 396.669,Z 637.859,A -85,B 0,C 180,E1 18203.471,E2 18203.471} C_VEL
LIN {X 0,Y 393.121,Z 656.739,A -85,B 0,C 180,E1 18201.721,E2 18201.721} C_VEL
LIN {X 0,Y 389.523,Z 674.038,A -85,B 0,C 180,E1 18199.807,E2 18199.807} C_VEL
LIN {X 0,Y 385.997,Z 689.913,A -85,B 0,C 180,E1 18197.721,E2 18197.721} C_VEL
LIN {X 0,Y 382.408,Z 705.437,A -85,B 0,C 180,E1 18195.314,E2 18195.314} C_VEL
LIN {X 0,Y 379.194,Z 719.161,A -85,B 0,C 180,E1 18192.798,E2 18192.798} C_VEL
LIN {X 0,Y 376.288,Z 731.482,A -85,B 0,C 180,E1 18190.102,E2 18190.102} C_VEL
LIN {X 0,Y 373.665,Z 743.048,A -85,B 0,C 180,E1 18187.072,E2 18187.072} C_VEL
LIN {X 0,Y 371.662,Z 752.703,A -85,B 0,C 180,E1 18184.013,E2 18184.013} C_VEL
LIN {X 0,Y 370.156,Z 760.994,A -85,B 0,C 180,E1 18180.776,E2 18180.776} C_VEL
LIN {X 0,Y 369.148,Z 767.453,A -85,B 0,C 180,E1 18177.518,E2 18177.518} C_VEL
LIN {X 0,Y 368.562,Z 772.526,A -85,B 0,C 180,E1 18174.085,E2 18174.085} C_VEL
LIN {X 0,Y 368.286,Z 775.862,A -85,B 0,C 180,E1 18170.785,E2 18170.785} C_VEL
LIN {X 0,Y 368.174,Z 777.539,A -85,B 0,C 180,E1 18167.614,E2 18167.614} C_VEL
LIN {X 0,Y 368.156,Z 777.842,A -85,B 0,C 180,E1 18164.244,E2 18164.244} C_VEL
LIN {X 0,Y 368.18,Z 776.77,A -85,B 0,C 180,E1 18161.148,E2 18161.148} C_VEL
LIN {X 0,Y 368.296,Z 774.074,A -85,B 0,C 180,E1 18157.833,E2 18157.833} C_VEL
LIN {X 0,Y 368.632,Z 769.767,A -85,B 0,C 180,E1 18154.455,E2 18154.455} C_VEL
LIN {X 0,Y 369.291,Z 763.994,A -85,B 0,C 180,E1 18151.191,E2 18151.191} C_VEL
LIN {X 0,Y 370.372,Z 756.521,A -85,B 0,C 180,E1 18147.961,E2 18147.961} C_VEL
LIN {X 0,Y 372.032,Z 747.159,A -85,B 0,C 180,E1 18144.706,E2 18144.706} C_VEL
LIN {X 0,Y 374.159,Z 736.612,A -85,B 0,C 180,E1 18141.69,E2 18141.69} C_VEL
LIN {X 0,Y 376.78,Z 724.334,A -85,B 0,C 180,E1 18138.79,E2 18138.79} C_VEL
LIN {X 0,Y 379.843,Z 710.56,A -85,B 0,C 180,E1 18136.057,E2 18136.057} C_VEL
LIN {X 0,Y 383.36,Z 694.853,A -85,B 0,C 180,E1 18133.43,E2 18133.43} C_VEL
LIN {X 0,Y 386.935,Z 678.732,A -85,B 0,C 180,E1 18131.151,E2 18131.151} C_VEL
LIN {X 0,Y 390.476,Z 661.623,A -85,B 0,C 180,E1 18129.121,E2 18129.121} C_VEL
LIN {X 0,Y 394.198,Z 642.464,A -85,B 0,C 180,E1 18127.214,E2 18127.214} C_VEL
LIN {X 0,Y 397.497,Z 623.932,A -85,B 0,C 180,E1 18125.667,E2 18125.667} C_VEL
LIN {X 0,Y 400.593,Z 603.981,A -85,B 0,C 180,E1 18124.3,E2 18124.3} C_VEL
LIN {X 0,Y 403.34,Z 583.153,A -85,B 0,C 180,E1 18123.149,E2 18123.149} C_VEL
LIN {X 0,Y 405.76,Z 560.88,A -85,B 0,C 180,E1 18122.193,E2 18122.193} C_VEL
LIN {X 0,Y 407.553,Z 539.252,A -85,B 0,C 180,E1 18121.509,E2 18121.509} C_VEL
LIN {X 0,Y 411.937,Z 448.406,A -85,B 0,C 180,E1 18119.627,E2 18119.627} C_VEL
LIN {X 0,Y 417.662,Z 335.451,A -85,B 0,C 180,E1 18117.288,E2 18117.288} C_VEL
LIN {X 0,Y 404.748,Z 316.026,A -85,B 0,C 180,E1 18114.852,E2 18114.852} C_VEL
LIN {X 0,Y 392.141,Z 298.053,A -85,B 0,C 180,E1 18112.256,E2 18112.256} C_VEL
LIN {X 0,Y 384.583,Z 287.771,A -85,B 0,C 180,E1 18110.588,E2 18110.588} C_VEL
LIN {X 0,Y 380.825,Z 282.706,A -85,B 0,C 180,E1 18109.718,E2 18109.718} C_VEL
LIN {X 0,Y 377.122,Z 277.665,A -85,B 0,C 180,E1 18108.835,E2 18108.835} C_VEL
LIN {X 0,Y 374.305,Z 273.971,A -85,B 0,C 180,E1 18108.153,E2 18108.153} C_VEL
LIN {X 0,Y 373.472,Z 272.513,A -85,B 0,C 180,E1 18107.933,E2 18107.933} C_VEL
LIN {X 0,Y 370.877,Z 269.907,A -85,B 0,C 180,E1 18107.313,E2 18107.313} C_VEL
LIN {X 0,Y 369.745,Z 266.675,A -85,B 0,C 180,E1 18106.942,E2 18106.942} C_VEL
LIN {X 0,Y 369.743,Z 266.677,A -85,B 0,C 180,E1 18102.813,E2 18102.813} C_VEL
LIN {X 0,Y 369.739,Z 266.672,A -85,B 0,C 180,E1 18098.712,E2 18098.712} C_VEL
LIN {X 0,Y 369.735,Z 266.672,A -85,B 0,C 180,E1 18094.655,E2 18094.655} C_VEL
LIN {X 0,Y 369.733,Z 266.672,A -85,B 0,C 180,E1 18094.621,E2 18094.621} C_VEL
LIN {X 0,Y 368.693,Z 266.81,A -85,B 0,C 180,E1 18093.427,E2 18093.427} C_VEL
LIN {X 0,Y 362.179,Z 267.613,A -85,B 0,C 180,E1 18089.969,E2 18089.969} C_VEL
LIN {X 0,Y 361.785,Z 267.656,A -85,B 0,C 180,E1 18089.175,E2 18089.175} C_VEL
LIN {X 0,Y 361.785,Z 267.654,A -85,B 0,C 180,E1 18085.087,E2 18085.087} C_VEL
LIN {X 0,Y 361.781,Z 267.66,A -85,B 0,C 180,E1 18081.098,E2 18081.098} C_VEL
LIN {X 0,Y 361.788,Z 267.664,A -85,B 0,C 180,E1 18076.904,E2 18076.904} C_VEL
LIN {X 0,Y 361.789,Z 267.666,A -85,B 0,C 180,E1 18072.802,E2 18072.802} C_VEL
LIN {X 0,Y 361.8,Z 267.666,A -85,B 0,C 180,E1 18068.607,E2 18068.607} C_VEL
LIN {X 0,Y 361.795,Z 267.667,A -85,B 0,C 180,E1 18064.463,E2 18064.463} C_VEL
LIN {X 0,Y 361.806,Z 267.665,A -85,B 0,C 180,E1 18060.354,E2 18060.354} C_VEL
LIN {X 0,Y 361.789,Z 267.665,A -85,B 0,C 180,E1 18056.258,E2 18056.258} C_VEL
LIN {X 0,Y 361.793,Z 267.663,A -85,B 0,C 180,E1 18052.158,E2 18052.158} C_VEL
LIN {X 0,Y 361.787,Z 267.663,A -85,B 0,C 180,E1 18048.019,E2 18048.019} C_VEL
LIN {X 0,Y 361.774,Z 267.664,A -85,B 0,C 180,E1 18043.838,E2 18043.838} C_VEL
LIN {X 0,Y 361.773,Z 267.663,A -85,B 0,C 180,E1 18039.799,E2 18039.799} C_VEL
LIN {X 0,Y 361.782,Z 267.665,A -85,B 0,C 180,E1 18035.863,E2 18035.863} C_VEL
LIN {X 0,Y 361.77,Z 267.669,A -85,B 0,C 180,E1 18031.673,E2 18031.673} C_VEL
LIN {X 0,Y 361.775,Z 267.672,A -85,B 0,C 180,E1 18027.663,E2 18027.663} C_VEL
LIN {X 0,Y 361.774,Z 267.673,A -85,B 0,C 180,E1 18023.622,E2 18023.622} C_VEL
LIN {X 0,Y 361.769,Z 267.673,A -85,B 0,C 180,E1 18019.535,E2 18019.535} C_VEL
LIN {X 0,Y 361.76,Z 267.671,A -85,B 0,C 180,E1 18015.384,E2 18015.384} C_VEL
LIN {X 0,Y 361.756,Z 267.668,A -85,B 0,C 180,E1 18011.315,E2 18011.315} C_VEL
LIN {X 0,Y 361.758,Z 267.667,A -85,B 0,C 180,E1 18007.302,E2 18007.302} C_VEL
LIN {X 0,Y 361.751,Z 267.671,A -85,B 0,C 180,E1 18003.167,E2 18003.167} C_VEL
LIN {X 0,Y 361.751,Z 267.676,A -85,B 0,C 180,E1 17999.048,E2 17999.048} C_VEL
LIN {X 0,Y 361.747,Z 267.668,A -85,B 0,C 180,E1 17994.924,E2 17994.924} C_VEL
LIN {X 0,Y 361.754,Z 267.671,A -85,B 0,C 180,E1 17990.934,E2 17990.934} C_VEL
LIN {X 0,Y 361.759,Z 267.67,A -85,B 0,C 180,E1 17986.899,E2 17986.899} C_VEL
LIN {X 0,Y 361.767,Z 267.668,A -85,B 0,C 180,E1 17982.963,E2 17982.963} C_VEL
LIN {X 0,Y 361.771,Z 267.664,A -85,B 0,C 180,E1 17978.942,E2 17978.942} C_VEL
LIN {X 0,Y 361.779,Z 267.665,A -85,B 0,C 180,E1 17974.984,E2 17974.984} C_VEL
LIN {X 0,Y 361.757,Z 267.757,A -85,B 0,C 180,E1 17973.992,E2 17973.992} C_VEL
LIN {X 0,Y 363.119,Z 271.185,A -85,B 0,C 180,E1 17973.153,E2 17973.153} C_VEL
LIN {X 0,Y 364.422,Z 273.227,A -85,B 0,C 180,E1 17972.551,E2 17972.551} C_VEL
LIN {X 0,Y 366.24,Z 276.707,A -85,B 0,C 180,E1 17971.637,E2 17971.637} C_VEL
LIN {X 0,Y 371.595,Z 286.918,A -85,B 0,C 180,E1 17969.073,E2 17969.073} C_VEL
LIN {X 0,Y 373.204,Z 289.857,A -85,B 0,C 180,E1 17968.458,E2 17968.458} C_VEL
LIN {X 0,Y 383.839,Z 305.283,A -85,B 0,C 180,E1 17965.849,E2 17965.849} C_VEL
LIN {X 0,Y 396.685,Z 325.077,A -85,B 0,C 180,E1 17962.956,E2 17962.956} C_VEL
LIN {X 0,Y 409.427,Z 346.038,A -85,B 0,C 180,E1 17960.311,E2 17960.311} C_VEL
LIN {X 0,Y 413.678,Z 353.825,A -85,B 0,C 180,E1 17959.472,E2 17959.472} C_VEL
LIN {X 0,Y 403.213,Z 548.034,A -85,B 0,C 180,E1 17955.4,E2 17955.4} C_VEL
LIN {X 0,Y 400.399,Z 602.02,A -85,B 0,C 180,E1 17954.234,E2 17954.234} C_VEL
LIN {X 0,Y 398.123,Z 624.911,A -85,B 0,C 180,E1 17953.523,E2 17953.523} C_VEL
LIN {X 0,Y 395.276,Z 646.911,A -85,B 0,C 180,E1 17952.58,E2 17952.58} C_VEL
LIN {X 0,Y 391.964,Z 668.94,A -85,B 0,C 180,E1 17951.349,E2 17951.349} C_VEL
LIN {X 0,Y 388.472,Z 689.223,A -85,B 0,C 180,E1 17949.942,E2 17949.942} C_VEL
LIN {X 0,Y 384.592,Z 709.467,A -85,B 0,C 180,E1 17948.222,E2 17948.222} C_VEL
LIN {X 0,Y 380.712,Z 728.495,A -85,B 0,C 180,E1 17946.266,E2 17946.266} C_VEL
LIN {X 0,Y 376.745,Z 746.982,A -85,B 0,C 180,E1 17944.005,E2 17944.005} C_VEL
LIN {X 0,Y 373.26,Z 763.177,A -85,B 0,C 180,E1 17941.668,E2 17941.668} C_VEL
LIN {X 0,Y 369.81,Z 779.068,A -85,B 0,C 180,E1 17938.942,E2 17938.942} C_VEL
LIN {X 0,Y 366.982,Z 792.607,A -85,B 0,C 180,E1 17936.19,E2 17936.19} C_VEL
LIN {X 0,Y 364.506,Z 805.513,A -85,B 0,C 180,E1 17933.093,E2 17933.093} C_VEL
LIN {X 0,Y 362.664,Z 816.57,A -85,B 0,C 180,E1 17929.924,E2 17929.924} C_VEL
LIN {X 0,Y 361.393,Z 825.677,A -85,B 0,C 180,E1 17926.721,E2 17926.721} C_VEL
LIN {X 0,Y 360.612,Z 833.138,A -85,B 0,C 180,E1 17923.466,E2 17923.466} C_VEL
LIN {X 0,Y 360.241,Z 838.938,A -85,B 0,C 180,E1 17920.23,E2 17920.23} C_VEL
LIN {X 0,Y 360.144,Z 842.973,A -85,B 0,C 180,E1 17917.015,E2 17917.015} C_VEL
LIN {X 0,Y 360.142,Z 845.526,A -85,B 0,C 180,E1 17913.819,E2 17913.819} C_VEL
LIN {X 0,Y 360.179,Z 846.428,A -85,B 0,C 180,E1 17910.794,E2 17910.794} C_VEL
LIN {X 0,Y 360.18,Z 845.932,A -85,B 0,C 180,E1 17907.612,E2 17907.612} C_VEL
LIN {X 0,Y 360.176,Z 843.934,A -85,B 0,C 180,E1 17904.583,E2 17904.583} C_VEL
LIN {X 0,Y 360.209,Z 840.332,A -85,B 0,C 180,E1 17901.378,E2 17901.378} C_VEL
LIN {X 0,Y 360.421,Z 835.342,A -85,B 0,C 180,E1 17898.315,E2 17898.315} C_VEL
LIN {X 0,Y 360.928,Z 828.369,A -85,B 0,C 180,E1 17895.069,E2 17895.069} C_VEL
LIN {X 0,Y 361.845,Z 819.889,A -85,B 0,C 180,E1 17891.908,E2 17891.908} C_VEL
LIN {X 0,Y 363.207,Z 809.787,A -85,B 0,C 180,E1 17888.86,E2 17888.86} C_VEL
LIN {X 0,Y 365.15,Z 797.518,A -85,B 0,C 180,E1 17885.748,E2 17885.748} C_VEL
LIN {X 0,Y 367.602,Z 783.705,A -85,B 0,C 180,E1 17882.803,E2 17882.803} C_VEL
LIN {X 0,Y 370.4,Z 768.791,A -85,B 0,C 180,E1 17880.128,E2 17880.128} C_VEL
LIN {X 0,Y 373.796,Z 751.418,A -85,B 0,C 180,E1 17877.475,E2 17877.475} C_VEL
LIN {X 0,Y 377.466,Z 732.579,A -85,B 0,C 180,E1 17875.046,E2 17875.046} C_VEL
LIN {X 0,Y 381.271,Z 712.855,A -85,B 0,C 180,E1 17872.902,E2 17872.902} C_VEL
LIN {X 0,Y 385.186,Z 691.713,A -85,B 0,C 180,E1 17870.987,E2 17870.987} C_VEL
LIN {X 0,Y 388.862,Z 670.804,A -85,B 0,C 180,E1 17869.418,E2 17869.418} C_VEL
LIN {X 0,Y 392.614,Z 647.886,A -85,B 0,C 180,E1 17867.998,E2 17867.998} C_VEL
LIN {X 0,Y 396.215,Z 624.263,A -85,B 0,C 180,E1 17866.84,E2 17866.84} C_VEL
LIN {X 0,Y 399.579,Z 598.845,A -85,B 0,C 180,E1 17865.891,E2 17865.891} C_VEL
LIN {X 0,Y 402.315,Z 569.591,A -85,B 0,C 180,E1 17865.066,E2 17865.066} C_VEL
LIN {X 0,Y 408.768,Z 498.325,A -85,B 0,C 180,E1 17863.209,E2 17863.209} C_VEL
LIN {X 0,Y 417.062,Z 429.148,A -85,B 0,C 180,E1 17861.297,E2 17861.297} C_VEL
LIN {X 0,Y 426.989,Z 363.514,A -85,B 0,C 180,E1 17859.437,E2 17859.437} C_VEL
LIN {X 0,Y 428.44,Z 354.48,A -85,B 0,C 180,E1 17859.154,E2 17859.154} C_VEL
LIN {X 0,Y 428.244,Z 348.895,A -85,B 0,C 180,E1 17858.054,E2 17858.054} C_VEL
LIN {X 0,Y 428.512,Z 344.946,A -85,B 0,C 180,E1 17856.847,E2 17856.847} C_VEL
LIN {X 0,Y 429.031,Z 343.657,A -85,B 0,C 180,E1 17855.925,E2 17855.925} C_VEL
LIN {X 0,Y 429.431,Z 345.789,A -85,B 0,C 180,E1 17854.957,E2 17854.957} C_VEL
LIN {X 0,Y 429.458,Z 346.522,A -85,B 0,C 180,E1 17854.825,E2 17854.825} C_VEL
LIN {X 0,Y 418.553,Z 413.345,A -85,B 0,C 180,E1 17852.931,E2 17852.931} C_VEL
LIN {X 0,Y 410.258,Z 477.386,A -85,B 0,C 180,E1 17851.146,E2 17851.146} C_VEL
LIN {X 0,Y 402.876,Z 552.783,A -85,B 0,C 180,E1 17849.103,E2 17849.103} C_VEL
LIN {X 0,Y 400.537,Z 574.739,A -85,B 0,C 180,E1 17848.264,E2 17848.264} C_VEL
LIN {X 0,Y 397.792,Z 595.761,A -85,B 0,C 180,E1 17847.225,E2 17847.225} C_VEL
LIN {X 0,Y 394.379,Z 617.734,A -85,B 0,C 180,E1 17845.855,E2 17845.855} C_VEL
LIN {X 0,Y 390.655,Z 638.444,A -85,B 0,C 180,E1 17844.256,E2 17844.256} C_VEL
LIN {X 0,Y 386.912,Z 657.296,A -85,B 0,C 180,E1 17842.488,E2 17842.488} C_VEL
LIN {X 0,Y 382.841,Z 675.772,A -85,B 0,C 180,E1 17840.407,E2 17840.407} C_VEL
LIN {X 0,Y 379.005,Z 691.954,A -85,B 0,C 180,E1 17838.219,E2 17838.219} C_VEL
LIN {X 0,Y 375.237,Z 707.281,A -85,B 0,C 180,E1 17835.773,E2 17835.773} C_VEL
LIN {X 0,Y 371.674,Z 721.555,A -85,B 0,C 180,E1 17833.062,E2 17833.062} C_VEL
LIN {X 0,Y 368.511,Z 734.334,A -85,B 0,C 180,E1 17830.16,E2 17830.16} C_VEL
LIN {X 0,Y 365.923,Z 745.012,A -85,B 0,C 180,E1 17827.223,E2 17827.223} C_VEL
LIN {X 0,Y 363.737,Z 754.853,A -85,B 0,C 180,E1 17823.943,E2 17823.943} C_VEL
LIN {X 0,Y 362.259,Z 762.531,A -85,B 0,C 180,E1 17820.793,E2 17820.793} C_VEL
LIN {X 0,Y 361.219,Z 768.85,A -85,B 0,C 180,E1 17817.464,E2 17817.464} C_VEL
LIN {X 0,Y 360.629,Z 773.547,A -85,B 0,C 180,E1 17814.114,E2 17814.114} C_VEL
LIN {X 0,Y 360.329,Z 776.764,A -85,B 0,C 180,E1 17810.741,E2 17810.741} C_VEL
LIN {X 0,Y 360.213,Z 778.373,A -85,B 0,C 180,E1 17807.498,E2 17807.498} C_VEL
LIN {X 0,Y 360.191,Z 778.583,A -85,B 0,C 180,E1 17804.217,E2 17804.217} C_VEL
LIN {X 0,Y 360.218,Z 777.486,A -85,B 0,C 180,E1 17801.052,E2 17801.052} C_VEL
LIN {X 0,Y 360.338,Z 774.911,A -85,B 0,C 180,E1 17797.832,E2 17797.832} C_VEL
LIN {X 0,Y 360.672,Z 770.927,A -85,B 0,C 180,E1 17794.555,E2 17794.555} C_VEL
LIN {X 0,Y 361.317,Z 765.381,A -85,B 0,C 180,E1 17791.311,E2 17791.311} C_VEL
LIN {X 0,Y 362.418,Z 758.117,A -85,B 0,C 180,E1 17788.018,E2 17788.018} C_VEL
LIN {X 0,Y 364.062,Z 749.232,A -85,B 0,C 180,E1 17784.782,E2 17784.782} C_VEL
LIN {X 0,Y 366.215,Z 738.857,A -85,B 0,C 180,E1 17781.705,E2 17781.705} C_VEL
LIN {X 0,Y 368.835,Z 727.104,A -85,B 0,C 180,E1 17778.8,E2 17778.8} C_VEL
LIN {X 0,Y 371.991,Z 713.563,A -85,B 0,C 180,E1 17775.979,E2 17775.979} C_VEL
LIN {X 0,Y 375.49,Z 698.713,A -85,B 0,C 180,E1 17773.373,E2 17773.373} C_VEL
LIN {X 0,Y 379.107,Z 682.834,A -85,B 0,C 180,E1 17771.041,E2 17771.041} C_VEL
LIN {X 0,Y 383.076,Z 664.672,A -85,B 0,C 180,E1 17768.788,E2 17768.788} C_VEL
LIN {X 0,Y 386.857,Z 646.233,A -85,B 0,C 180,E1 17766.87,E2 17766.87} C_VEL
LIN {X 0,Y 390.525,Z 626.633,A -85,B 0,C 180,E1 17765.176,E2 17765.176} C_VEL
LIN {X 0,Y 393.709,Z 607.121,A -85,B 0,C 180,E1 17763.792,E2 17763.792} C_VEL
LIN {X 0,Y 396.744,Z 585.482,A -85,B 0,C 180,E1 17762.548,E2 17762.548} C_VEL
LIN {X 0,Y 399.273,Z 563.652,A -85,B 0,C 180,E1 17761.571,E2 17761.571} C_VEL
LIN {X 0,Y 401.159,Z 542.007,A -85,B 0,C 180,E1 17760.862,E2 17760.862} C_VEL
LIN {X 0,Y 402.993,Z 508.551,A -85,B 0,C 180,E1 17760.119,E2 17760.119} C_VEL
LIN {X 0,Y 411.875,Z 339.095,A -85,B 0,C 180,E1 17756.571,E2 17756.571} C_VEL
LIN {X 0,Y 398.174,Z 318.475,A -85,B 0,C 180,E1 17753.907,E2 17753.907} C_VEL
LIN {X 0,Y 384.582,Z 299.235,A -85,B 0,C 180,E1 17751.002,E2 17751.002} C_VEL
LIN {X 0,Y 376.689,Z 288.689,A -85,B 0,C 180,E1 17749.177,E2 17749.177} C_VEL
LIN {X 0,Y 373.123,Z 283.871,A -85,B 0,C 180,E1 17748.314,E2 17748.314} C_VEL
LIN {X 0,Y 369.354,Z 278.816,A -85,B 0,C 180,E1 17747.366,E2 17747.366} C_VEL
LIN {X 0,Y 366.562,Z 275.174,A -85,B 0,C 180,E1 17746.644,E2 17746.644} C_VEL
LIN {X 0,Y 365.558,Z 273.51,A -85,B 0,C 180,E1 17746.364,E2 17746.364} C_VEL
LIN {X 0,Y 362.934,Z 270.92,A -85,B 0,C 180,E1 17745.706,E2 17745.706} C_VEL
LIN {X 0,Y 361.816,Z 267.808,A -85,B 0,C 180,E1 17745.334,E2 17745.334} C_VEL
LIN {X 0,Y 361.797,Z 267.661,A -85,B 0,C 180,E1 17741.156,E2 17741.156} C_VEL
LIN {X 0,Y 361.812,Z 267.666,A -85,B 0,C 180,E1 17736.986,E2 17736.986} C_VEL
LIN {X 0,Y 361.797,Z 267.657,A -85,B 0,C 180,E1 17732.694,E2 17732.694} C_VEL
LIN {X 0,Y 361.785,Z 267.656,A -85,B 0,C 180,E1 17729.175,E2 17729.175} C_VEL
LIN {X 0,Y 360.964,Z 267.766,A -85,B 0,C 180,E1 17728.041,E2 17728.041} C_VEL
LIN {X 0,Y 357.107,Z 268.245,A -85,B 0,C 180,E1 17726.082,E2 17726.082} C_VEL
LIN {X 0,Y 354.173,Z 268.613,A -85,B 0,C 180,E1 17724.332,E2 17724.332} C_VEL
LIN {X 0,Y 353.825,Z 268.656,A -85,B 0,C 180,E1 17723.609,E2 17723.609} C_VEL
LIN {X 0,Y 353.828,Z 268.656,A -85,B 0,C 180,E1 17719.418,E2 17719.418} C_VEL
LIN {X 0,Y 353.828,Z 268.655,A -85,B 0,C 180,E1 17715.268,E2 17715.268} C_VEL
LIN {X 0,Y 353.828,Z 268.656,A -85,B 0,C 180,E1 17711.19,E2 17711.19} C_VEL
LIN {X 0,Y 353.828,Z 268.656,A -85,B 0,C 180,E1 17707.05,E2 17707.05} C_VEL
LIN {X 0,Y 353.835,Z 268.657,A -85,B 0,C 180,E1 17702.881,E2 17702.881} C_VEL
LIN {X 0,Y 353.831,Z 268.662,A -85,B 0,C 180,E1 17698.863,E2 17698.863} C_VEL
LIN {X 0,Y 353.832,Z 268.664,A -85,B 0,C 180,E1 17694.746,E2 17694.746} C_VEL
LIN {X 0,Y 353.828,Z 268.665,A -85,B 0,C 180,E1 17690.732,E2 17690.732} C_VEL
LIN {X 0,Y 353.828,Z 268.663,A -85,B 0,C 180,E1 17686.635,E2 17686.635} C_VEL
LIN {X 0,Y 353.833,Z 268.66,A -85,B 0,C 180,E1 17682.478,E2 17682.478} C_VEL
LIN {X 0,Y 353.828,Z 268.654,A -85,B 0,C 180,E1 17678.435,E2 17678.435} C_VEL
LIN {X 0,Y 353.836,Z 268.649,A -85,B 0,C 180,E1 17674.213,E2 17674.213} C_VEL
LIN {X 0,Y 353.851,Z 268.647,A -85,B 0,C 180,E1 17670.006,E2 17670.006} C_VEL
LIN {X 0,Y 353.839,Z 268.647,A -85,B 0,C 180,E1 17665.793,E2 17665.793} C_VEL
LIN {X 0,Y 353.837,Z 268.651,A -85,B 0,C 180,E1 17661.622,E2 17661.622} C_VEL
LIN {X 0,Y 353.822,Z 268.655,A -85,B 0,C 180,E1 17657.427,E2 17657.427} C_VEL
LIN {X 0,Y 353.822,Z 268.657,A -85,B 0,C 180,E1 17653.396,E2 17653.396} C_VEL
LIN {X 0,Y 353.818,Z 268.664,A -85,B 0,C 180,E1 17649.267,E2 17649.267} C_VEL
LIN {X 0,Y 353.813,Z 268.664,A -85,B 0,C 180,E1 17645.186,E2 17645.186} C_VEL
LIN {X 0,Y 353.803,Z 268.657,A -85,B 0,C 180,E1 17640.969,E2 17640.969} C_VEL
LIN {X 0,Y 353.806,Z 268.66,A -85,B 0,C 180,E1 17636.92,E2 17636.92} C_VEL
LIN {X 0,Y 353.808,Z 268.664,A -85,B 0,C 180,E1 17632.855,E2 17632.855} C_VEL
LIN {X 0,Y 353.808,Z 268.657,A -85,B 0,C 180,E1 17628.754,E2 17628.754} C_VEL
LIN {X 0,Y 353.806,Z 268.662,A -85,B 0,C 180,E1 17624.593,E2 17624.593} C_VEL
LIN {X 0,Y 353.81,Z 268.658,A -85,B 0,C 180,E1 17620.519,E2 17620.519} C_VEL
LIN {X 0,Y 353.807,Z 268.656,A -85,B 0,C 180,E1 17616.289,E2 17616.289} C_VEL
LIN {X 0,Y 353.851,Z 268.88,A -85,B 0,C 180,E1 17615.633,E2 17615.633} C_VEL
LIN {X 0,Y 355.376,Z 272.489,A -85,B 0,C 180,E1 17614.679,E2 17614.679} C_VEL
LIN {X 0,Y 356.42,Z 273.851,A -85,B 0,C 180,E1 17614.218,E2 17614.218} C_VEL
LIN {X 0,Y 358.452,Z 277.84,A -85,B 0,C 180,E1 17613.134,E2 17613.134} C_VEL
LIN {X 0,Y 362.051,Z 284.884,A -85,B 0,C 180,E1 17611.279,E2 17611.279} C_VEL
LIN {X 0,Y 364.271,Z 288.669,A -85,B 0,C 180,E1 17610.345,E2 17610.345} C_VEL
LIN {X 0,Y 376.955,Z 307.143,A -85,B 0,C 180,E1 17607.036,E2 17607.036} C_VEL
LIN {X 0,Y 388.233,Z 324.338,A -85,B 0,C 180,E1 17604.382,E2 17604.382} C_VEL
LIN {X 0,Y 400.831,Z 344.733,A -85,B 0,C 180,E1 17601.646,E2 17601.646} C_VEL
LIN {X 0,Y 407.868,Z 357.19,A -85,B 0,C 180,E1 17600.201,E2 17600.201} C_VEL
LIN {X 0,Y 396.951,Z 550.966,A -85,B 0,C 180,E1 17596.081,E2 17596.081} C_VEL
LIN {X 0,Y 394.151,Z 601.685,A -85,B 0,C 180,E1 17594.961,E2 17594.961} C_VEL
LIN {X 0,Y 391.8,Z 624.538,A -85,B 0,C 180,E1 17594.242,E2 17594.242} C_VEL
LIN {X 0,Y 388.932,Z 645.897,A -85,B 0,C 180,E1 17593.319,E2 17593.319} C_VEL
LIN {X 0,Y 385.553,Z 667.645,A -85,B 0,C 180,E1 17592.103,E2 17592.103} C_VEL
LIN {X 0,Y 381.925,Z 688.081,A -85,B 0,C 180,E1 17590.68,E2 17590.68} C_VEL
LIN {X 0,Y 377.833,Z 708.59,A -85,B 0,C 180,E1 17588.92,E2 17588.92} C_VEL
LIN {X 0,Y 373.874,Z 727.177,A -85,B 0,C 180,E1 17586.991,E2 17586.991} C_VEL
LIN {X 0,Y 369.747,Z 745.701,A -85,B 0,C 180,E1 17584.706,E2 17584.706} C_VEL
